C03650=1118.505,289.970,-75.818,-178.026,10.350,149.542
C03651=1118.509,289.721,-75.787,-178.029,10.347,149.543
C03652=1118.513,289.474,-75.756,-178.032,10.345,149.543
C03653=1118.517,289.225,-75.725,-178.035,10.342,149.543
C03654=1118.521,288.978,-75.694,-178.038,10.340,149.543
C03655=1118.526,288.730,-75.664,-178.041,10.338,149.543
C03656=1118.530,288.482,-75.632,-178.044,10.335,149.544
C03657=1118.534,288.234,-75.601,-178.047,10.333,149.544
C03658=1118.538,287.985,-75.570,-178.050,10.330,149.544
C03659=1118.542,287.738,-75.540,-178.053,10.327,149.544
C03660=1118.547,287.490,-75.509,-178.056,10.325,149.544
C03661=1118.551,287.241,-75.478,-178.060,10.322,149.544
C03662=1118.554,286.994,-75.447,-178.062,10.319,149.544
C03663=1118.558,286.745,-75.416,-178.065,10.318,149.545
C03664=1118.563,286.497,-75.385,-178.068,10.315,149.545
C03665=1118.568,286.249,-75.354,-178.071,10.313,149.545
C03666=1118.571,286.001,-75.324,-178.074,10.310,149.545
C03667=1118.576,285.753,-75.293,-178.077,10.307,149.545
C03668=1118.580,285.505,-75.262,-178.081,10.305,149.546
C03669=1118.583,285.257,-75.232,-178.084,10.302,149.546
C03670=1118.588,285.009,-75.201,-178.087,10.299,149.546
C03671=1118.593,284.761,-75.170,-178.090,10.297,149.546
C03672=1118.596,284.512,-75.140,-178.093,10.295,149.546
C03673=1118.601,284.264,-75.109,-178.096,10.292,149.546
C03674=1118.605,284.016,-75.078,-178.098,10.290,149.547
C03675=1118.608,283.768,-75.048,-178.102,10.287,149.547
C03676=1118.613,283.520,-75.017,-178.105,10.284,149.547
C03677=1118.617,283.273,-74.987,-178.108,10.282,149.547
C03678=1118.621,283.025,-74.956,-178.111,10.279,149.547
C03679=1118.626,282.776,-74.925,-178.114,10.277,149.548
C03680=1118.629,282.528,-74.895,-178.117,10.274,149.548
C03681=1118.634,282.280,-74.864,-178.120,10.272,149.548
C03682=1118.638,282.031,-74.834,-178.123,10.270,149.548
C03683=1118.642,281.783,-74.803,-178.126,10.267,149.548
C03684=1118.646,281.536,-74.773,-178.129,10.264,149.548
C03685=1118.650,281.323,-74.747,-178.132,10.262,149.549
C03686=1118.653,281.110,-74.721,-178.134,10.260,149.549
C03687=1118.657,280.897,-74.694,-178.138,10.257,149.549
C03688=1118.661,280.684,-74.668,-178.140,10.255,149.549
C03689=1118.664,280.471,-74.642,-178.143,10.252,149.549
C03690=1118.668,280.258,-74.616,-178.146,10.251,149.549
C03691=1118.671,280.045,-74.591,-178.149,10.248,149.550
C03692=1118.675,279.832,-74.564,-178.152,10.245,149.550
C03693=1118.679,279.584,-74.534,-178.155,10.243,149.550
C03694=1118.684,279.336,-74.503,-178.158,10.240,149.550
C03695=1118.687,279.087,-74.473,-178.161,10.237,149.550
C03696=1118.692,278.839,-74.443,-178.164,10.235,149.550
C03697=1118.696,278.591,-74.412,-178.167,10.232,149.551
C03698=1118.700,278.343,-74.383,-178.170,10.230,149.551
C03699=1118.705,278.095,-74.352,-178.173,10.227,149.551
C03700=1118.708,277.847,-74.322,-178.176,10.224,149.551
C03701=1118.713,277.598,-74.292,-178.180,10.222,149.551
C03702=1118.717,277.351,-74.262,-178.183,10.219,149.551
C03703=1118.721,277.102,-74.232,-178.186,10.216,149.551
C03704=1118.726,276.854,-74.201,-178.189,10.214,149.552
C03705=1118.730,276.606,-74.172,-178.192,10.211,149.552
C03706=1118.734,276.358,-74.142,-178.195,10.208,149.552
C03707=1118.738,276.109,-74.111,-178.198,10.205,149.552
C03708=1118.742,275.861,-74.081,-178.202,10.202,149.552
C03709=1118.746,275.613,-74.052,-178.205,10.200,149.552
C03710=1118.751,275.365,-74.021,-178.208,10.197,149.553
C03711=1118.755,275.117,-73.991,-178.210,10.195,149.553
C03712=1118.759,274.869,-73.961,-178.213,10.192,149.553
C03713=1118.763,274.621,-73.932,-178.216,10.190,149.553
C03714=1118.767,274.373,-73.901,-178.219,10.187,149.553
C03715=1118.771,274.124,-73.871,-178.222,10.184,149.553
C03716=1118.775,273.876,-73.842,-178.225,10.181,149.553
C03717=1118.779,273.628,-73.812,-178.228,10.179,149.553
C03718=1118.784,273.380,-73.782,-178.231,10.176,149.554
C03719=1118.788,273.132,-73.751,-178.234,10.173,149.554
C03720=1118.792,272.884,-73.722,-178.237,10.171,149.554
C03721=1118.796,272.635,-73.692,-178.240,10.168,149.554
C03722=1118.800,272.387,-73.663,-178.243,10.165,149.554
C03723=1118.805,272.139,-73.632,-178.245,10.163,149.554
C03724=1118.809,271.891,-73.603,-178.248,10.161,149.554
C03725=1118.813,271.643,-73.573,-178.251,10.158,149.554
C03726=1118.817,271.395,-73.543,-178.254,10.155,149.555
C03727=1118.822,271.147,-73.514,-178.257,10.152,149.555
C03728=1118.826,270.898,-73.484,-178.260,10.149,149.555
C03729=1118.831,270.650,-73.454,-178.262,10.148,149.555
C03730=1118.835,270.402,-73.425,-178.265,10.145,149.555
C03731=1118.839,270.154,-73.395,-178.268,10.142,149.555
C03732=1118.843,269.906,-73.365,-178.271,10.139,149.555
C03733=1118.847,269.657,-73.336,-178.274,10.136,149.555
C03734=1118.851,269.409,-73.306,-178.276,10.134,149.555
C03735=1118.855,269.161,-73.277,-178.279,10.132,149.555
C03736=1118.860,268.913,-73.247,-178.282,10.129,149.556
C03737=1118.864,268.664,-73.217,-178.285,10.126,149.556
C03738=1118.868,268.416,-73.187,-178.287,10.124,149.556
C03739=1118.873,268.168,-73.158,-178.290,10.121,149.556
C03740=1118.877,267.920,-73.128,-178.293,10.119,149.556
C03741=1118.880,267.707,-73.103,-178.296,10.117,149.556
C03742=1118.884,267.493,-73.078,-178.298,10.115,149.556
C03743=1118.888,267.281,-73.052,-178.300,10.113,149.556
C03744=1118.891,267.068,-73.027,-178.302,10.110,149.556
C03745=1118.895,266.854,-73.002,-178.304,10.108,149.556
C03746=1118.898,266.641,-72.977,-178.307,10.106,149.557
C03747=1118.903,266.428,-72.952,-178.310,10.104,149.557
C03748=1118.906,266.215,-72.926,-178.312,10.102,149.557
C03749=1118.910,265.967,-72.897,-178.314,10.100,149.557
C03750=1118.914,265.719,-72.867,-178.317,10.097,149.557
C03751=1118.918,265.470,-72.838,-178.320,10.095,149.557
C03752=1118.923,265.222,-72.809,-178.323,10.092,149.557
C03753=1118.927,264.973,-72.779,-178.325,10.090,149.557
C03754=1118.931,264.725,-72.750,-178.328,10.088,149.557
C03755=1118.935,264.477,-72.721,-178.331,10.085,149.558
C03756=1118.940,264.229,-72.692,-178.334,10.082,149.558
C03757=1118.944,263.981,-72.662,-178.337,10.080,149.558
C03758=1118.949,263.733,-72.633,-178.341,10.076,149.558
C03759=1118.952,263.485,-72.604,-178.344,10.074,149.558
C03760=1118.956,263.236,-72.575,-178.347,10.071,149.558
C03761=1118.961,262.988,-72.546,-178.350,10.067,149.559
C03762=1118.965,262.739,-72.516,-178.354,10.065,149.559
C03763=1118.970,262.492,-72.487,-178.357,10.062,149.559
C03764=1118.974,262.243,-72.458,-178.360,10.059,149.559
C03765=1118.978,261.995,-72.429,-178.364,10.056,149.559
C03766=1118.982,261.746,-72.399,-178.367,10.054,149.559
C03767=1118.986,261.498,-72.371,-178.370,10.050,149.560
C03768=1118.991,261.250,-72.342,-178.373,10.047,149.560
C03769=1118.995,261.002,-72.313,-178.376,10.044,149.560
C03770=1118.999,260.754,-72.283,-178.379,10.042,149.560
C03771=1119.004,260.505,-72.254,-178.382,10.039,149.560
C03772=1119.007,260.257,-72.226,-178.386,10.036,149.560
C03773=1119.012,260.009,-72.197,-178.389,10.033,149.560
C03774=1119.017,259.760,-72.168,-178.392,10.030,149.560
C03775=1119.021,259.512,-72.138,-178.395,10.027,149.561
C03776=1119.025,259.263,-72.110,-178.398,10.025,149.561
C03777=1119.029,259.015,-72.081,-178.401,10.022,149.561
C03778=1119.033,258.768,-72.052,-178.404,10.019,149.561
C03779=1119.038,258.519,-72.023,-178.407,10.016,149.561
C03780=1119.041,258.271,-71.994,-178.410,10.013,149.561
C03781=1119.046,258.022,-71.965,-178.413,10.010,149.561
C03782=1119.051,257.774,-71.936,-178.416,10.007,149.561
C03783=1119.054,257.526,-71.908,-178.418,10.004,149.561
C03784=1119.059,257.277,-71.879,-178.421,10.002,149.561
C03785=1119.064,257.029,-71.850,-178.424,9.999,149.561
C03786=1119.067,256.781,-71.822,-178.427,9.996,149.562
C03787=1119.072,256.532,-71.793,-178.430,9.993,149.561
C03788=1119.076,256.284,-71.764,-178.432,9.991,149.562
C03789=1119.080,256.036,-71.735,-178.435,9.988,149.562
C03790=1119.085,255.787,-71.707,-178.436,9.986,149.561
C03791=1119.088,255.539,-71.679,-178.437,9.985,149.561
C03792=1119.093,255.291,-71.649,-178.438,9.983,149.561
C03793=1119.098,255.042,-71.621,-178.439,9.981,149.561
C03794=1119.101,254.794,-71.592,-178.441,9.980,149.561
C03795=1119.106,254.546,-71.564,-178.442,9.977,149.561
C03796=1119.110,254.298,-71.535,-178.444,9.976,149.561
C03797=1119.114,254.084,-71.510,-178.445,9.974,149.561
C03798=1119.118,253.872,-71.485,-178.447,9.972,149.561
C03799=1119.121,253.658,-71.462,-178.449,9.971,149.561
C03800=1119.125,253.445,-71.437,-178.450,9.970,149.561
C03801=1119.129,253.231,-71.412,-178.452,9.967,149.561
C03802=1119.132,253.019,-71.388,-178.454,9.965,149.561
C03803=1119.136,252.805,-71.363,-178.457,9.963,149.561
C03804=1119.140,252.591,-71.338,-178.459,9.961,149.562
C03805=1119.144,252.344,-71.310,-178.461,9.959,149.562
C03806=1119.148,252.095,-71.281,-178.464,9.957,149.562
C03807=1119.153,251.847,-71.253,-178.468,9.954,149.562
C03808=1119.157,251.598,-71.225,-178.471,9.951,149.562
C03809=1119.161,251.350,-71.196,-178.474,9.949,149.563
C03810=1119.166,251.102,-71.167,-178.477,9.946,149.563
C03811=1119.169,250.854,-71.139,-178.481,9.943,149.563
C03812=1119.174,250.605,-71.110,-178.484,9.941,149.563
C03813=1119.178,250.357,-71.083,-178.488,9.937,149.564
C03814=1119.183,250.108,-71.054,-178.492,9.934,149.564
C03815=1119.187,249.860,-71.026,-178.496,9.931,149.564
C03816=1119.190,249.612,-70.997,-178.500,9.928,149.564
C03817=1119.196,249.364,-70.969,-178.504,9.924,149.564
C03818=1119.199,249.115,-70.941,-178.509,9.920,149.565
C03819=1119.204,248.866,-70.912,-178.513,9.917,149.565
C03820=1119.208,248.619,-70.884,-178.518,9.913,149.565
C03821=1119.212,248.370,-70.856,-178.523,9.909,149.566
C03822=1119.217,248.122,-70.828,-178.528,9.904,149.566
C03823=1119.221,247.873,-70.800,-178.533,9.900,149.566
C03824=1119.225,247.625,-70.772,-178.538,9.896,149.567
C03825=1119.230,247.376,-70.744,-178.542,9.892,149.567
C03826=1119.234,247.128,-70.716,-178.543,9.890,149.567
C03827=1119.238,246.879,-70.688,-178.545,9.887,149.567
C03828=1119.243,246.631,-70.660,-178.547,9.885,149.566
C03829=1119.247,246.383,-70.631,-178.549,9.883,149.566
C03830=1119.251,246.135,-70.604,-178.551,9.880,149.566
C03831=1119.255,245.886,-70.576,-178.553,9.878,149.566
C03832=1119.260,245.637,-70.548,-178.554,9.875,149.566
C03833=1119.264,245.389,-70.520,-178.557,9.872,149.566
C03834=1119.268,245.141,-70.492,-178.559,9.870,149.566
C03835=1119.273,244.893,-70.464,-178.561,9.868,149.566
C03836=1119.277,244.644,-70.435,-178.563,9.866,149.566
C03837=1119.282,244.396,-70.408,-178.565,9.863,149.566
C03838=1119.286,244.147,-70.380,-178.567,9.861,149.566
C03839=1119.290,243.899,-70.352,-178.569,9.858,149.566
C03840=1119.295,243.650,-70.324,-178.571,9.856,149.566
C03841=1119.299,243.402,-70.296,-178.573,9.853,149.566
C03842=1119.303,243.153,-70.268,-178.575,9.851,149.566
C03843=1119.307,242.905,-70.241,-178.578,9.848,149.566
C03844=1119.312,242.658,-70.213,-178.580,9.846,149.566
C03845=1119.316,242.408,-70.185,-178.582,9.844,149.566
C03846=1119.321,242.160,-70.157,-178.584,9.841,149.566
C03847=1119.325,241.912,-70.129,-178.587,9.839,149.566
C03848=1119.329,241.663,-70.102,-178.589,9.836,149.566
C03849=1119.334,241.415,-70.074,-178.591,9.834,149.566
C03850=1119.337,241.167,-70.046,-178.594,9.831,149.566
C03851=1119.342,240.918,-70.019,-178.596,9.829,149.566
C03852=1119.346,240.669,-69.990,-178.598,9.826,149.566
C03853=1119.350,240.456,-69.967,-178.601,9.824,149.566
C03854=1119.354,240.243,-69.943,-178.603,9.822,149.566
C03855=1119.357,240.029,-69.919,-178.605,9.820,149.566
C03856=1119.361,239.816,-69.895,-178.607,9.818,149.566
C03857=1119.365,239.603,-69.872,-178.609,9.816,149.566
C03858=1119.368,239.389,-69.848,-178.611,9.813,149.566
C03859=1119.372,239.176,-69.824,-178.613,9.811,149.566
C03860=1119.376,238.963,-69.801,-178.615,9.809,149.566
C03861=1119.381,238.714,-69.773,-178.618,9.807,149.566
C03862=1119.385,238.466,-69.745,-178.621,9.804,149.567
C03863=1119.390,238.217,-69.718,-178.624,9.802,149.567
C03864=1119.393,237.969,-69.690,-178.625,9.799,149.567
C03865=1119.398,237.720,-69.663,-178.628,9.796,149.567
C03866=1119.402,237.472,-69.635,-178.631,9.794,149.567
C03867=1119.406,237.223,-69.608,-178.634,9.792,149.567
C03868=1119.411,236.975,-69.581,-178.637,9.789,149.567
C03869=1119.415,236.727,-69.553,-178.639,9.786,149.567
C03870=1119.420,236.478,-69.526,-178.642,9.783,149.567
C03871=1119.424,236.230,-69.498,-178.644,9.781,149.567
C03872=1119.428,235.981,-69.470,-178.647,9.778,149.567
C03873=1119.433,235.733,-69.443,-178.650,9.776,149.568
C03874=1119.437,235.484,-69.415,-178.653,9.773,149.568
C03875=1119.442,235.236,-69.388,-178.656,9.770,149.568
C03876=1119.445,234.988,-69.362,-178.659,9.767,149.568
C03877=1119.450,234.740,-69.334,-178.662,9.764,149.568
C03878=1119.454,234.491,-69.307,-178.665,9.762,149.568
C03879=1119.459,234.242,-69.279,-178.667,9.759,149.568
C03880=1119.463,233.994,-69.252,-178.670,9.756,149.568
C03881=1119.468,233.746,-69.225,-178.673,9.753,149.568
C03882=1119.472,233.496,-69.197,-178.676,9.751,149.568
C03883=1119.476,233.248,-69.170,-178.679,9.748,149.569
C03884=1119.481,233.000,-69.142,-178.682,9.745,149.569
C03885=1119.485,232.752,-69.116,-178.685,9.742,149.569
C03886=1119.489,232.503,-69.088,-178.688,9.740,149.569
C03887=1119.493,232.254,-69.061,-178.691,9.736,149.569
C03888=1119.498,232.006,-69.034,-178.694,9.733,149.569
C03889=1119.503,231.757,-69.007,-178.697,9.730,149.569
C03890=1119.507,231.509,-68.980,-178.700,9.727,149.569
C03891=1119.510,231.260,-68.953,-178.704,9.724,149.569
C03892=1119.515,231.012,-68.926,-178.707,9.721,149.569
C03893=1119.520,230.763,-68.899,-178.710,9.718,149.570
C03894=1119.524,230.515,-68.872,-178.713,9.715,149.570
C03895=1119.528,230.267,-68.845,-178.716,9.712,149.570
C03896=1119.533,230.018,-68.818,-178.720,9.709,149.570
C03897=1119.537,229.770,-68.791,-178.723,9.706,149.570
C03898=1119.541,229.521,-68.763,-178.726,9.702,149.570
C03899=1119.545,229.272,-68.737,-178.729,9.699,149.570
C03900=1119.550,229.024,-68.710,-178.732,9.696,149.570
C03901=1119.555,228.775,-68.683,-178.735,9.693,149.570
C03902=1119.559,228.527,-68.656,-178.739,9.689,149.570
C03903=1119.563,228.279,-68.629,-178.741,9.686,149.570
C03904=1119.568,228.030,-68.602,-178.744,9.684,149.571
C03905=1119.573,227.782,-68.575,-178.748,9.680,149.571
C03906=1119.576,227.533,-68.548,-178.750,9.677,149.571
C03907=1119.581,227.284,-68.521,-178.754,9.673,149.571
C03908=1119.585,227.036,-68.496,-178.757,9.670,149.571
C03909=1119.589,226.823,-68.472,-178.759,9.668,149.571
C03910=1119.593,226.609,-68.449,-178.762,9.664,149.571
C03911=1119.597,226.395,-68.427,-178.764,9.662,149.571
C03912=1119.600,226.182,-68.403,-178.767,9.659,149.571
C03913=1119.604,225.969,-68.380,-178.769,9.656,149.571
C03914=1119.608,225.755,-68.358,-178.771,9.654,149.571
C03915=1119.612,225.542,-68.335,-178.774,9.651,149.571
C03916=1119.615,225.329,-68.312,-178.777,9.648,149.571
C03917=1119.620,225.079,-68.285,-178.779,9.645,149.571
C03918=1119.624,224.831,-68.259,-178.782,9.642,149.571
C03919=1119.628,224.582,-68.231,-178.785,9.639,149.571
C03920=1119.632,224.334,-68.205,-178.788,9.635,149.571
C03921=1119.637,224.085,-68.179,-178.790,9.632,149.571
C03922=1119.641,223.837,-68.152,-178.793,9.629,149.571
C03923=1119.646,223.588,-68.125,-178.796,9.626,149.571
C03924=1119.650,223.339,-68.099,-178.798,9.623,149.571
C03925=1119.655,223.091,-68.072,-178.802,9.619,149.571
C03926=1119.659,222.843,-68.046,-178.804,9.616,149.570
C03927=1119.664,222.594,-68.020,-178.807,9.613,149.570
C03928=1119.668,222.346,-67.993,-178.809,9.610,149.570
C03929=1119.673,222.097,-67.967,-178.812,9.607,149.570
C03930=1119.677,221.849,-67.941,-178.814,9.604,149.570
C03931=1119.682,221.600,-67.914,-178.817,9.601,149.570
C03932=1119.686,221.351,-67.888,-178.819,9.598,149.570
C03933=1119.690,221.103,-67.862,-178.822,9.594,149.570
C03934=1119.695,220.854,-67.835,-178.824,9.591,149.570
C03935=1119.699,220.606,-67.809,-178.827,9.588,149.570
C03936=1119.704,220.357,-67.782,-178.829,9.585,149.570
C03937=1119.708,220.108,-67.756,-178.832,9.582,149.570
C03938=1119.712,219.860,-67.730,-178.834,9.578,149.569
C03939=1119.717,219.611,-67.704,-178.837,9.575,149.569
C03940=1119.721,219.363,-67.677,-178.839,9.572,149.569
C03941=1119.725,219.114,-67.651,-178.842,9.569,149.569
C03942=1119.730,218.866,-67.625,-178.844,9.567,149.569
C03943=1119.734,218.617,-67.599,-178.846,9.564,149.569
C03944=1119.739,218.368,-67.573,-178.848,9.560,149.569
C03945=1119.743,218.120,-67.546,-178.851,9.557,149.569
C03946=1119.748,217.871,-67.520,-178.853,9.554,149.569
C03947=1119.751,217.623,-67.494,-178.855,9.552,149.569
C03948=1119.756,217.374,-67.468,-178.857,9.548,149.568
C03949=1119.761,217.125,-67.442,-178.860,9.545,149.568
C03950=1119.765,216.877,-67.415,-178.862,9.543,149.568
C03951=1119.769,216.629,-67.390,-178.864,9.539,149.568
C03952=1119.774,216.379,-67.364,-178.866,9.536,149.568
C03953=1119.779,216.131,-67.338,-178.868,9.534,149.568
C03954=1119.782,215.883,-67.311,-178.871,9.531,149.568
C03955=1119.787,215.634,-67.286,-178.873,9.527,149.568
C03956=1119.792,215.385,-67.259,-178.875,9.525,149.568
C03957=1119.796,215.136,-67.234,-178.877,9.522,149.568
C03958=1119.800,214.888,-67.207,-178.879,9.519,149.567
C03959=1119.805,214.639,-67.182,-178.881,9.516,149.567
C03960=1119.809,214.391,-67.156,-178.883,9.513,149.567
C03961=1119.814,214.142,-67.130,-178.885,9.510,149.567
C03962=1119.819,213.893,-67.104,-178.887,9.508,149.567
C03963=1119.823,213.645,-67.078,-178.889,9.505,149.567
C03964=1119.827,213.396,-67.052,-178.891,9.502,149.567
C03965=1119.831,213.114,-67.023,-178.894,9.499,149.567
C03966=1119.838,212.832,-66.994,-178.896,9.496,149.566
C03967=1119.842,212.550,-66.964,-178.899,9.493,149.566
C03968=1119.847,212.267,-66.935,-178.902,9.489,149.566
C03969=1119.851,212.019,-66.909,-178.904,9.487,149.566
C03970=1119.856,211.770,-66.883,-178.906,9.483,149.566
C03971=1119.861,211.521,-66.857,-178.909,9.480,149.566
C03972=1119.865,211.272,-66.832,-178.911,9.478,149.566
C03973=1119.870,211.024,-66.806,-178.913,9.475,149.566
C03974=1119.874,210.775,-66.780,-178.916,9.472,149.566
C03975=1119.878,210.526,-66.755,-178.919,9.469,149.566
C03976=1119.882,210.278,-66.729,-178.921,9.467,149.566
C03977=1119.887,210.030,-66.704,-178.923,9.464,149.566
C03978=1119.891,209.781,-66.678,-178.926,9.461,149.566
C03979=1119.896,209.532,-66.652,-178.929,9.458,149.566
C03980=1119.900,209.284,-66.627,-178.931,9.455,149.566
C03981=1119.905,209.035,-66.601,-178.933,9.453,149.566
C03982=1119.909,208.786,-66.575,-178.936,9.450,149.566
C03983=1119.914,208.538,-66.550,-178.939,9.447,149.566
C03984=1119.918,208.289,-66.524,-178.941,9.444,149.566
C03985=1119.925,207.896,-66.483,-178.946,9.439,149.566
C03986=1119.932,207.502,-66.442,-178.950,9.435,149.566
C03987=1119.940,207.108,-66.403,-178.955,9.430,149.567
C03988=1119.947,206.715,-66.362,-178.959,9.426,149.567
C03989=1119.951,206.466,-66.336,-178.962,9.423,149.567
C03990=1119.956,206.218,-66.311,-178.964,9.420,149.567
C03991=1119.960,205.969,-66.286,-178.967,9.417,149.567
C03992=1119.964,205.720,-66.261,-178.970,9.414,149.567
C03993=1119.969,205.472,-66.235,-178.973,9.412,149.567
C03994=1119.973,205.223,-66.209,-178.976,9.409,149.567
C03995=1119.977,204.973,-66.184,-178.979,9.406,149.567
C03996=1119.982,204.725,-66.159,-178.982,9.403,149.567
C03997=1119.987,204.477,-66.133,-178.985,9.400,149.568
C03998=1119.992,204.228,-66.109,-178.987,9.397,149.568
C03999=1119.996,203.979,-66.083,-178.990,9.394,149.568
C04000=1120.000,203.731,-66.058,-178.993,9.392,149.568
C04001=1120.004,203.482,-66.033,-178.997,9.388,149.568
C04002=1120.009,203.233,-66.007,-178.999,9.385,149.568
C04003=1120.014,202.985,-65.982,-179.002,9.382,149.568
C04004=1120.018,202.735,-65.957,-179.005,9.380,149.568
C04005=1120.023,202.487,-65.931,-179.008,9.377,149.568
C04006=1120.027,202.238,-65.907,-179.012,9.373,149.568
C04007=1120.032,201.990,-65.882,-179.014,9.370,149.568
C04008=1120.036,201.741,-65.857,-179.017,9.368,149.569
C04009=1120.041,201.493,-65.831,-179.021,9.364,149.569
C04010=1120.045,201.243,-65.807,-179.024,9.361,149.569
C04011=1120.049,200.995,-65.781,-179.026,9.359,149.569
C04012=1120.054,200.746,-65.756,-179.030,9.355,149.569
C04013=1120.058,200.497,-65.731,-179.033,9.352,149.569
C04014=1120.063,200.249,-65.707,-179.036,9.349,149.569
C04015=1120.067,200.000,-65.681,-179.039,9.346,149.569
C04016=1120.072,199.751,-65.656,-179.042,9.343,149.569
C04017=1120.076,199.537,-65.635,-179.045,9.340,149.569
C04018=1120.080,199.324,-65.614,-179.048,9.337,149.570
C04019=1120.083,199.110,-65.592,-179.050,9.334,149.570
C04020=1120.087,198.896,-65.571,-179.053,9.331,149.570
C04021=1120.091,198.683,-65.549,-179.056,9.328,149.570
C04022=1120.095,198.469,-65.528,-179.059,9.325,149.570
C04023=1120.098,198.255,-65.506,-179.061,9.323,149.570
C04024=1120.103,198.042,-65.485,-179.064,9.319,149.570
C04025=1120.107,197.793,-65.460,-179.067,9.317,149.570
C04026=1120.111,197.544,-65.436,-179.071,9.313,149.570
C04027=1120.116,197.295,-65.411,-179.074,9.309,149.570
C04028=1120.120,197.047,-65.386,-179.077,9.306,149.570
C04029=1120.125,196.798,-65.361,-179.080,9.303,149.570
C04030=1120.130,196.549,-65.336,-179.083,9.299,149.570
C04031=1120.134,196.301,-65.312,-179.087,9.295,149.570
C04032=1120.138,196.051,-65.287,-179.088,9.293,149.570
C04033=1120.143,195.803,-65.263,-179.090,9.290,149.570
C04034=1120.148,195.555,-65.237,-179.092,9.288,149.570
C04035=1120.151,195.306,-65.213,-179.093,9.285,149.570
C04036=1120.157,195.057,-65.188,-179.096,9.282,149.570
C04037=1120.160,194.808,-65.164,-179.097,9.279,149.569
C04038=1120.166,194.559,-65.139,-179.099,9.277,149.569
C04039=1120.170,194.311,-65.115,-179.101,9.275,149.569
C04040=1120.174,194.061,-65.090,-179.103,9.271,149.569
C04041=1120.179,193.813,-65.066,-179.105,9.269,149.569
C04042=1120.184,193.565,-65.041,-179.107,9.266,149.569
C04043=1120.187,193.316,-65.016,-179.109,9.263,149.569
C04044=1120.193,193.067,-64.992,-179.111,9.261,149.569
C04045=1120.197,192.818,-64.967,-179.113,9.259,149.569
C04046=1120.202,192.569,-64.942,-179.115,9.255,149.568
C04047=1120.206,192.321,-64.918,-179.117,9.253,149.568
C04048=1120.210,192.072,-64.894,-179.119,9.250,149.568
C04049=1120.215,191.823,-64.869,-179.121,9.247,149.568
C04050=1120.219,191.574,-64.845,-179.123,9.245,149.568
C04051=1120.224,191.326,-64.821,-179.125,9.242,149.568
C04052=1120.228,191.077,-64.796,-179.127,9.239,149.568
C04053=1120.233,190.828,-64.772,-179.129,9.237,149.568
C04054=1120.238,190.579,-64.747,-179.132,9.234,149.568
C04055=1120.242,190.331,-64.723,-179.133,9.231,149.568
C04056=1120.247,190.082,-64.698,-179.136,9.228,149.568
C04057=1120.251,189.833,-64.674,-179.138,9.226,149.568
C04058=1120.256,189.584,-64.651,-179.140,9.223,149.568
C04059=1120.261,189.335,-64.626,-179.142,9.220,149.568
C04060=1120.265,189.086,-64.602,-179.145,9.217,149.568
C04061=1120.269,188.838,-64.578,-179.147,9.214,149.568
C04062=1120.274,188.589,-64.553,-179.149,9.212,149.568
C04063=1120.278,188.340,-64.528,-179.152,9.209,149.568
C04064=1120.282,188.092,-64.504,-179.154,9.206,149.568
C04065=1120.288,187.842,-64.480,-179.156,9.203,149.567
C04066=1120.292,187.594,-64.456,-179.159,9.200,149.567
C04067=1120.297,187.345,-64.432,-179.161,9.198,149.567
C04068=1120.301,187.096,-64.407,-179.163,9.195,149.567
C04069=1120.306,186.848,-64.383,-179.166,9.192,149.567
C04070=1120.310,186.599,-64.360,-179.167,9.189,149.567
C04071=1120.315,186.350,-64.336,-179.170,9.186,149.567
C04072=1120.319,186.101,-64.311,-179.173,9.183,149.567
C04073=1120.323,185.887,-64.291,-179.174,9.181,149.567
C04074=1120.327,185.674,-64.270,-179.176,9.179,149.567
C04075=1120.331,185.459,-64.249,-179.179,9.175,149.567
C04076=1120.335,185.246,-64.228,-179.181,9.173,149.567
C04077=1120.338,185.032,-64.208,-179.183,9.171,149.567
C04078=1120.343,184.818,-64.187,-179.186,9.168,149.567
C04079=1120.347,184.604,-64.166,-179.187,9.166,149.567
C04080=1120.350,184.390,-64.146,-179.189,9.163,149.567
C04081=1120.355,184.142,-64.122,-179.192,9.160,149.567
C04082=1120.360,183.893,-64.097,-179.194,9.157,149.567
C04083=1120.364,183.644,-64.074,-179.197,9.154,149.567
C04084=1120.368,183.395,-64.050,-179.200,9.151,149.567
C04085=1120.373,183.146,-64.026,-179.202,9.148,149.567
C04086=1120.377,182.898,-64.002,-179.205,9.145,149.567
C04087=1120.382,182.649,-63.978,-179.207,9.142,149.567
C04088=1120.387,182.400,-63.955,-179.210,9.139,149.567
C04089=1120.392,182.152,-63.930,-179.213,9.136,149.567
C04090=1120.396,181.902,-63.907,-179.215,9.133,149.567
C04091=1120.400,181.653,-63.882,-179.218,9.130,149.567
C04092=1120.405,181.404,-63.859,-179.221,9.126,149.567
C04093=1120.409,181.156,-63.835,-179.224,9.123,149.567
C04094=1120.414,180.907,-63.811,-179.226,9.120,149.567
C04095=1120.418,180.658,-63.787,-179.229,9.117,149.567
C04096=1120.423,180.409,-63.764,-179.231,9.114,149.567
C04097=1120.427,180.161,-63.740,-179.234,9.110,149.567
C04098=1120.432,179.912,-63.717,-179.237,9.107,149.567
C04099=1120.437,179.663,-63.693,-179.240,9.104,149.567
C04100=1120.441,179.415,-63.669,-179.242,9.101,149.567
C04101=1120.446,179.166,-63.646,-179.245,9.098,149.567
C04102=1120.451,178.916,-63.622,-179.247,9.094,149.567
C04103=1120.454,178.667,-63.598,-179.250,9.091,149.566
C04104=1120.459,178.418,-63.575,-179.251,9.089,149.566
C04105=1120.464,178.170,-63.551,-179.254,9.085,149.566
C04106=1120.468,177.921,-63.527,-179.255,9.083,149.566
C04107=1120.473,177.672,-63.504,-179.258,9.080,149.566
C04108=1120.478,177.423,-63.480,-179.260,9.076,149.566
C04109=1120.482,177.174,-63.456,-179.262,9.074,149.566
C04110=1120.487,176.925,-63.433,-179.264,9.071,149.566
C04111=1120.491,176.676,-63.410,-179.267,9.067,149.566
C04112=1120.496,176.428,-63.386,-179.268,9.065,149.566
C04113=1120.501,176.179,-63.362,-179.271,9.062,149.566
C04114=1120.504,175.930,-63.339,-179.273,9.058,149.565
C04115=1120.509,175.681,-63.316,-179.275,9.056,149.565
C04116=1120.514,175.432,-63.293,-179.277,9.053,149.565
C04117=1120.518,175.184,-63.269,-179.280,9.050,149.565
C04118=1120.523,174.935,-63.245,-179.281,9.047,149.565
C04119=1120.528,174.686,-63.222,-179.284,9.044,149.565
C04120=1120.532,174.437,-63.199,-179.286,9.041,149.565
C04121=1120.537,174.188,-63.175,-179.288,9.038,149.565
C04122=1120.542,173.940,-63.153,-179.290,9.035,149.565
C04123=1120.546,173.691,-63.129,-179.293,9.032,149.565
C04124=1120.551,173.442,-63.105,-179.294,9.029,149.564
C04125=1120.555,173.193,-63.082,-179.297,9.026,149.564
C04126=1120.560,172.944,-63.059,-179.300,9.023,149.564
C04127=1120.565,172.695,-63.035,-179.302,9.020,149.564
C04128=1120.569,172.446,-63.013,-179.304,9.017,149.564
C04129=1120.573,172.232,-62.992,-179.305,9.015,149.564
C04130=1120.576,172.018,-62.972,-179.308,9.012,149.564
C04131=1120.581,171.804,-62.953,-179.309,9.009,149.564
C04132=1120.585,171.590,-62.933,-179.311,9.007,149.564
C04133=1120.589,171.377,-62.913,-179.313,9.005,149.564
C04134=1120.593,171.163,-62.893,-179.316,9.001,149.564
C04135=1120.597,170.948,-62.872,-179.317,8.999,149.563
C04136=1120.601,170.734,-62.853,-179.319,8.996,149.563
C04137=1120.605,170.485,-62.830,-179.322,8.993,149.563
C04138=1120.609,170.236,-62.807,-179.324,8.990,149.563
C04139=1120.615,169.988,-62.784,-179.326,8.987,149.563
C04140=1120.619,169.739,-62.761,-179.328,8.984,149.563
C04141=1120.624,169.490,-62.737,-179.331,8.981,149.563
C04142=1120.628,169.241,-62.714,-179.333,8.978,149.563
C04143=1120.633,168.992,-62.691,-179.335,8.975,149.563
C04144=1120.637,168.743,-62.668,-179.337,8.972,149.563
C04145=1120.641,168.495,-62.645,-179.339,8.969,149.562
C04146=1120.647,168.246,-62.622,-179.342,8.966,149.562
C04147=1120.652,167.997,-62.599,-179.344,8.963,149.562
C04148=1120.656,167.748,-62.577,-179.346,8.960,149.562
C04149=1120.660,167.499,-62.553,-179.348,8.957,149.562
C04150=1120.665,167.250,-62.530,-179.351,8.954,149.562
C04151=1120.670,167.002,-62.507,-179.353,8.951,149.562
C04152=1120.675,166.752,-62.485,-179.355,8.947,149.562
C04153=1120.679,166.503,-62.462,-179.358,8.944,149.562
C04154=1120.683,166.254,-62.439,-179.360,8.942,149.562
C04155=1120.688,166.005,-62.415,-179.362,8.938,149.561
C04156=1120.693,165.757,-62.394,-179.364,8.935,149.561
C04157=1120.697,165.508,-62.370,-179.367,8.932,149.561
C04158=1120.701,165.259,-62.348,-179.369,8.928,149.561
C04159=1120.706,165.010,-62.324,-179.372,8.925,149.561
C04160=1120.711,164.761,-62.303,-179.374,8.922,149.561
C04161=1120.716,164.512,-62.279,-179.376,8.919,149.561
C04162=1120.720,164.263,-62.256,-179.379,8.916,149.561
C04163=1120.725,164.014,-62.234,-179.381,8.913,149.561
C04164=1120.730,163.766,-62.211,-179.383,8.910,149.560
C04165=1120.734,163.517,-62.188,-179.385,8.907,149.560
C04166=1120.739,163.267,-62.165,-179.388,8.904,149.560
C04167=1120.743,163.018,-62.143,-179.390,8.900,149.560
C04168=1120.748,162.770,-62.121,-179.392,8.897,149.560
C04169=1120.752,162.521,-62.098,-179.395,8.894,149.560
C04170=1120.757,162.271,-62.075,-179.397,8.890,149.560
C04171=1120.761,162.022,-62.052,-179.399,8.887,149.560
C04172=1120.766,161.774,-62.030,-179.401,8.884,149.560
C04173=1120.771,161.525,-62.007,-179.404,8.881,149.560
C04174=1120.775,161.276,-61.984,-179.407,8.878,149.560
C04175=1120.781,161.027,-61.962,-179.409,8.874,149.559
C04176=1120.785,160.778,-61.939,-179.411,8.871,149.559
C04177=1120.789,160.529,-61.917,-179.413,8.868,149.559
C04178=1120.794,160.281,-61.894,-179.416,8.864,149.559
C04179=1120.798,160.031,-61.872,-179.418,8.861,149.559
C04180=1120.803,159.782,-61.850,-179.420,8.858,149.559
C04181=1120.808,159.534,-61.827,-179.423,8.855,149.559
C04182=1120.812,159.284,-61.805,-179.425,8.851,149.558
C04183=1120.817,159.035,-61.782,-179.427,8.848,149.558
C04184=1120.822,158.787,-61.760,-179.430,8.845,149.558
C04185=1120.826,158.572,-61.741,-179.431,8.842,149.558
C04186=1120.830,158.358,-61.722,-179.434,8.839,149.558
C04187=1120.834,158.145,-61.702,-179.435,8.837,149.558
C04188=1120.838,157.930,-61.683,-179.438,8.833,149.558
C04189=1120.842,157.716,-61.664,-179.439,8.831,149.558
C04190=1120.846,157.502,-61.645,-179.442,8.828,149.558
C04191=1120.850,157.288,-61.626,-179.444,8.824,149.558
C04192=1120.853,157.075,-61.607,-179.446,8.822,149.557
C04193=1120.858,156.825,-61.584,-179.448,8.819,149.557
C04194=1120.863,156.576,-61.562,-179.451,8.815,149.557
C04195=1120.867,156.327,-61.540,-179.453,8.812,149.557
C04196=1120.872,156.078,-61.517,-179.456,8.808,149.557
C04197=1120.877,155.829,-61.495,-179.458,8.805,149.557
C04198=1120.881,155.580,-61.473,-179.460,8.801,149.557
C04199=1120.886,155.331,-61.451,-179.462,8.798,149.556
C04200=1120.890,155.082,-61.429,-179.465,8.795,149.556
C04201=1120.896,154.834,-61.406,-179.467,8.791,149.556
C04202=1120.900,154.584,-61.384,-179.470,8.788,149.556
C04203=1120.905,154.336,-61.363,-179.472,8.784,149.556
C04204=1120.909,154.086,-61.341,-179.475,8.781,149.556
C04205=1120.914,153.838,-61.319,-179.477,8.777,149.556
C04206=1120.919,153.588,-61.296,-179.479,8.774,149.555
C04207=1120.924,153.339,-61.275,-179.481,8.771,149.555
C04208=1120.928,153.091,-61.252,-179.484,8.766,149.555
C04209=1120.932,152.842,-61.230,-179.487,8.763,149.555
C04210=1120.937,152.593,-61.208,-179.489,8.760,149.555
C04211=1120.942,152.344,-61.186,-179.491,8.756,149.555
C04212=1120.946,152.095,-61.164,-179.494,8.752,149.554
C04213=1120.952,151.846,-61.142,-179.496,8.749,149.554
C04214=1120.956,151.596,-61.120,-179.498,8.745,149.554
C04215=1120.961,151.348,-61.098,-179.501,8.742,149.554
C04216=1120.965,151.099,-61.076,-179.503,8.738,149.554
C04217=1120.970,150.850,-61.055,-179.505,8.734,149.554
C04218=1120.974,150.601,-61.033,-179.508,8.731,149.553
C04219=1120.979,150.352,-61.011,-179.511,8.727,149.553
C04220=1120.983,150.103,-60.989,-179.513,8.724,149.553
C04221=1120.988,149.853,-60.968,-179.515,8.720,149.553
C04222=1120.993,149.605,-60.946,-179.518,8.716,149.553
C04223=1120.998,149.355,-60.924,-179.520,8.713,149.553
C04224=1121.002,149.107,-60.902,-179.522,8.709,149.552
C04225=1121.007,148.857,-60.880,-179.525,8.705,149.552
C04226=1121.012,148.609,-60.859,-179.527,8.702,149.552
C04227=1121.016,148.360,-60.837,-179.529,8.698,149.552
C04228=1121.021,148.110,-60.816,-179.532,8.694,149.552
C04229=1121.026,147.861,-60.794,-179.534,8.691,149.551
C04230=1121.030,147.612,-60.772,-179.537,8.686,149.551
C04231=1121.035,147.363,-60.750,-179.539,8.683,149.551
C04232=1121.040,147.115,-60.729,-179.542,8.679,149.551
C04233=1121.044,146.865,-60.707,-179.544,8.675,149.550
C04234=1121.049,146.616,-60.686,-179.546,8.672,149.550
C04235=1121.054,146.368,-60.664,-179.549,8.667,149.550
C04236=1121.058,146.118,-60.642,-179.551,8.664,149.550
C04237=1121.063,145.869,-60.621,-179.553,8.660,149.549
C04238=1121.068,145.621,-60.600,-179.556,8.657,149.549
C04239=1121.072,145.371,-60.578,-179.559,8.652,149.549
C04240=1121.077,145.122,-60.557,-179.561,8.649,149.549
C04241=1121.081,144.908,-60.538,-179.562,8.646,149.548
C04242=1121.085,144.694,-60.520,-179.563,8.643,149.548
C04243=1121.090,144.480,-60.501,-179.564,8.640,149.548
C04244=1121.093,144.265,-60.483,-179.566,8.637,149.548
C04245=1121.097,144.051,-60.464,-179.568,8.634,149.547
C04246=1121.101,143.837,-60.446,-179.569,8.631,149.547
C04247=1121.106,143.623,-60.428,-179.570,8.628,149.547
C04248=1121.109,143.409,-60.409,-179.572,8.625,149.546
C04249=1121.114,143.160,-60.388,-179.573,8.622,149.546
C04250=1121.118,142.911,-60.366,-179.575,8.619,149.546
C04251=1121.124,142.661,-60.345,-179.576,8.615,149.545
C04252=1121.128,142.413,-60.324,-179.577,8.612,149.545
C04253=1121.133,142.164,-60.303,-179.579,8.609,149.545
C04254=1121.137,141.915,-60.281,-179.581,8.605,149.544
C04255=1121.142,141.665,-60.260,-179.583,8.602,149.544
C04256=1121.147,141.417,-60.239,-179.584,8.598,149.544
C04257=1121.151,141.167,-60.218,-179.586,8.595,149.543
C04258=1121.156,140.918,-60.196,-179.587,8.592,149.543
C04259=1121.161,140.669,-60.175,-179.589,8.588,149.543
C04260=1121.166,140.420,-60.154,-179.590,8.585,149.542
C04261=1121.170,140.172,-60.133,-179.592,8.582,149.542
C04262=1121.175,139.922,-60.111,-179.593,8.578,149.542
C04263=1121.180,139.673,-60.090,-179.595,8.575,149.541
C04264=1121.184,139.424,-60.070,-179.597,8.572,149.541
C04265=1121.189,139.175,-60.048,-179.598,8.569,149.541
C04266=1121.194,138.925,-60.027,-179.600,8.565,149.541
C04267=1121.198,138.677,-60.006,-179.601,8.562,149.540
C04268=1121.203,138.428,-59.985,-179.603,8.559,149.540
C04269=1121.208,138.179,-59.964,-179.605,8.555,149.539
C04270=1121.212,137.930,-59.943,-179.606,8.552,149.539
C04271=1121.217,137.680,-59.921,-179.608,8.548,149.539
C04272=1121.222,137.431,-59.900,-179.609,8.545,149.539
C04273=1121.226,137.183,-59.879,-179.611,8.542,149.538
C04274=1121.231,136.933,-59.858,-179.612,8.539,149.538
C04275=1121.236,136.684,-59.838,-179.614,8.535,149.538
C04276=1121.241,136.436,-59.816,-179.617,8.532,149.537
C04277=1121.245,136.186,-59.795,-179.618,8.529,149.537
C04278=1121.250,135.937,-59.775,-179.620,8.525,149.537
C04279=1121.255,135.688,-59.754,-179.621,8.522,149.536
C04280=1121.259,135.439,-59.732,-179.623,8.519,149.536
C04281=1121.264,135.190,-59.712,-179.625,8.515,149.536
C04282=1121.269,134.941,-59.691,-179.626,8.512,149.535
C04283=1121.274,134.692,-59.670,-179.628,8.509,149.535
C04284=1121.279,134.443,-59.648,-179.629,8.506,149.535
C04285=1121.283,134.194,-59.628,-179.631,8.502,149.535
C04286=1121.288,133.944,-59.607,-179.633,8.499,149.534
C04287=1121.292,133.695,-59.586,-179.634,8.496,149.534
C04288=1121.297,133.446,-59.565,-179.636,8.492,149.534
C04289=1121.302,133.197,-59.545,-179.638,8.488,149.533
C04290=1121.307,132.948,-59.523,-179.640,8.486,149.533
C04291=1121.311,132.700,-59.503,-179.641,8.482,149.533
C04292=1121.316,132.450,-59.482,-179.643,8.479,149.533
C04293=1121.321,132.201,-59.462,-179.645,8.476,149.532
C04294=1121.326,131.952,-59.441,-179.646,8.472,149.532
C04295=1121.330,131.703,-59.420,-179.648,8.469,149.532
C04296=1121.335,131.453,-59.399,-179.650,8.466,149.531
C04297=1121.339,131.239,-59.382,-179.651,8.463,149.531
C04298=1121.343,131.025,-59.364,-179.653,8.460,149.531
C04299=1121.348,130.811,-59.346,-179.654,8.457,149.531
C04300=1121.351,130.596,-59.328,-179.655,8.454,149.530
C04301=1121.356,130.382,-59.311,-179.657,8.451,149.530
C04302=1121.359,130.168,-59.293,-179.659,8.448,149.530
C04303=1121.363,129.953,-59.275,-179.660,8.445,149.530
C04304=1121.368,129.739,-59.257,-179.662,8.443,149.529
C04305=1121.372,129.490,-59.237,-179.664,8.439,149.529
C04306=1121.378,129.241,-59.216,-179.665,8.436,149.529
C04307=1121.382,128.992,-59.195,-179.667,8.433,149.529
C04308=1121.386,128.743,-59.175,-179.669,8.429,149.528
C04309=1121.392,128.494,-59.154,-179.670,8.426,149.528
C04310=1121.396,128.245,-59.134,-179.672,8.423,149.528
C04311=1121.400,127.996,-59.113,-179.673,8.420,149.527
C04312=1121.406,127.747,-59.092,-179.675,8.416,149.527
C04313=1121.410,127.498,-59.072,-179.678,8.413,149.527
C04314=1121.415,127.249,-59.051,-179.679,8.409,149.527
C04315=1121.420,127.000,-59.031,-179.681,8.406,149.526
C04316=1121.424,126.750,-59.011,-179.683,8.403,149.526
C04317=1121.429,126.501,-58.991,-179.685,8.399,149.526
C04318=1121.434,126.252,-58.970,-179.686,8.396,149.525
C04319=1121.438,126.003,-58.949,-179.688,8.393,149.525
C04320=1121.443,125.754,-58.929,-179.690,8.389,149.525
C04321=1121.448,125.505,-58.908,-179.691,8.386,149.525
C04322=1121.453,125.255,-58.888,-179.693,8.383,149.524
C04323=1121.457,125.006,-58.868,-179.695,8.379,149.524
C04324=1121.462,124.757,-58.847,-179.696,8.376,149.524
C04325=1121.467,124.508,-58.827,-179.698,8.373,149.524
C04326=1121.472,124.258,-58.807,-179.701,8.369,149.523
C04327=1121.476,124.010,-58.787,-179.702,8.366,149.523
C04328=1121.481,123.761,-58.766,-179.704,8.363,149.523
C04329=1121.486,123.512,-58.746,-179.706,8.359,149.523
C04330=1121.491,123.262,-58.726,-179.708,8.356,149.522
C04331=1121.495,123.013,-58.706,-179.709,8.353,149.522
C04332=1121.500,122.765,-58.685,-179.711,8.349,149.522
C04333=1121.505,122.515,-58.665,-179.713,8.346,149.521
C04334=1121.510,122.266,-58.645,-179.715,8.342,149.521
C04335=1121.514,122.017,-58.624,-179.716,8.339,149.521
C04336=1121.519,121.767,-58.604,-179.718,8.336,149.521
C04337=1121.523,121.518,-58.584,-179.720,8.332,149.520
C04338=1121.528,121.270,-58.564,-179.722,8.329,149.520
C04339=1121.533,121.020,-58.544,-179.724,8.326,149.520
C04340=1121.538,120.771,-58.523,-179.725,8.322,149.519
C04341=1121.543,120.522,-58.504,-179.727,8.319,149.519
C04342=1121.548,120.273,-58.483,-179.729,8.315,149.519
C04343=1121.552,120.024,-58.463,-179.731,8.312,149.519
C04344=1121.557,119.774,-58.443,-179.733,8.309,149.519
C04345=1121.562,119.526,-58.423,-179.734,8.305,149.518
C04346=1121.567,119.276,-58.404,-179.737,8.301,149.518
C04347=1121.571,119.027,-58.383,-179.738,8.299,149.518
C04348=1121.576,118.778,-58.364,-179.740,8.295,149.517
C04349=1121.581,118.529,-58.343,-179.742,8.292,149.517
C04350=1121.586,118.279,-58.323,-179.744,8.288,149.517
C04351=1121.591,118.031,-58.303,-179.745,8.285,149.517
C04352=1121.595,117.781,-58.283,-179.747,8.282,149.516
C04353=1121.599,117.567,-58.266,-179.749,8.278,149.516
C04354=1121.604,117.352,-58.249,-179.751,8.275,149.516
C04355=1121.607,117.139,-58.232,-179.752,8.273,149.516
C04356=1121.611,116.924,-58.215,-179.754,8.270,149.515
C04357=1121.615,116.710,-58.198,-179.756,8.266,149.515
C04358=1121.619,116.495,-58.181,-179.757,8.264,149.515
C04359=1121.624,116.281,-58.163,-179.758,8.261,149.515
C04360=1121.628,116.067,-58.147,-179.760,8.257,149.514
C04361=1121.633,115.817,-58.127,-179.762,8.254,149.514
C04362=1121.637,115.568,-58.106,-179.764,8.251,149.514
C04363=1121.642,115.318,-58.087,-179.766,8.247,149.514
C04364=1121.647,115.070,-58.068,-179.767,8.244,149.513
C04365=1121.652,114.821,-58.047,-179.769,8.240,149.513
C04366=1121.657,114.571,-58.028,-179.771,8.237,149.513
C04367=1121.662,114.322,-58.008,-179.773,8.234,149.513
C04368=1121.666,114.073,-57.988,-179.774,8.230,149.512
C04369=1121.671,113.824,-57.968,-179.777,8.226,149.512
C04370=1121.676,113.574,-57.949,-179.779,8.223,149.512
C04371=1121.680,113.326,-57.930,-179.781,8.219,149.511
C04372=1121.685,113.077,-57.909,-179.782,8.216,149.511
C04373=1121.690,112.827,-57.890,-179.784,8.212,149.511
C04374=1121.695,112.578,-57.871,-179.786,8.209,149.511
C04375=1121.700,112.329,-57.851,-179.788,8.206,149.510
C04376=1121.704,112.080,-57.831,-179.789,8.202,149.510
C04377=1121.709,111.831,-57.811,-179.792,8.198,149.510
C04378=1121.714,111.581,-57.792,-179.794,8.195,149.509
C04379=1121.719,111.332,-57.772,-179.796,8.191,149.509
C04380=1121.724,111.083,-57.753,-179.797,8.188,149.509
C04381=1121.728,110.834,-57.734,-179.799,8.184,149.509
C04382=1121.733,110.585,-57.713,-179.801,8.181,149.508
C04383=1121.738,110.336,-57.694,-179.804,8.176,149.508
C04384=1121.743,110.086,-57.674,-179.806,8.173,149.508
C04385=1121.748,109.837,-57.655,-179.809,8.169,149.508
C04386=1121.752,109.588,-57.636,-179.811,8.165,149.507
C04387=1121.757,109.338,-57.616,-179.813,8.162,149.507
C04388=1121.762,109.089,-57.597,-179.816,8.157,149.507
C04389=1121.767,108.840,-57.577,-179.818,8.154,149.507
C04390=1121.771,108.591,-57.558,-179.820,8.149,149.507
C04391=1121.776,108.342,-57.539,-179.822,8.146,149.506
C04392=1121.781,108.092,-57.519,-179.824,8.142,149.506
C04393=1121.786,107.843,-57.500,-179.827,8.138,149.506
C04394=1121.790,107.594,-57.481,-179.829,8.134,149.506
C04395=1121.795,107.345,-57.461,-179.831,8.131,149.505
C04396=1121.801,107.096,-57.442,-179.834,8.127,149.505
C04397=1121.805,106.847,-57.423,-179.836,8.123,149.505
C04398=1121.810,106.598,-57.404,-179.838,8.118,149.504
C04399=1121.815,106.348,-57.384,-179.840,8.115,149.504
C04400=1121.819,106.100,-57.365,-179.842,8.111,149.504
C04401=1121.824,105.849,-57.346,-179.845,8.107,149.504
C04402=1121.829,105.600,-57.327,-179.846,8.103,149.503
C04403=1121.834,105.351,-57.308,-179.848,8.100,149.503
C04404=1121.838,105.102,-57.288,-179.850,8.096,149.503
C04405=1121.844,104.853,-57.269,-179.853,8.092,149.502
C04406=1121.848,104.604,-57.250,-179.855,8.088,149.502
C04407=1121.853,104.354,-57.231,-179.857,8.084,149.502
C04408=1121.857,104.105,-57.212,-179.859,8.080,149.502
C04409=1121.862,103.890,-57.196,-179.860,8.077,149.501
C04410=1121.867,103.676,-57.179,-179.862,8.074,149.501
C04411=1121.870,103.462,-57.163,-179.864,8.070,149.501
C04412=1121.875,103.247,-57.146,-179.865,8.067,149.500
C04413=1121.879,103.033,-57.130,-179.867,8.063,149.500
C04414=1121.883,102.818,-57.114,-179.870,8.060,149.500
C04415=1121.887,102.603,-57.098,-179.871,8.057,149.500
C04416=1121.891,102.389,-57.081,-179.873,8.053,149.499
C04417=1121.896,102.141,-57.062,-179.874,8.049,149.499
C04418=1121.901,101.891,-57.043,-179.876,8.046,149.499
C04419=1121.906,101.642,-57.025,-179.878,8.041,149.498
C04420=1121.910,101.392,-57.005,-179.881,8.038,149.498
C04421=1121.915,101.143,-56.987,-179.882,8.034,149.498
C04422=1121.920,100.893,-56.967,-179.884,8.030,149.497
C04423=1121.925,100.645,-56.949,-179.886,8.027,149.497
C04424=1121.930,100.395,-56.930,-179.888,8.022,149.497
C04425=1121.934,100.146,-56.911,-179.890,8.018,149.496
C04426=1121.940,99.897,-56.892,-179.892,8.014,149.496
C04427=1121.944,99.647,-56.873,-179.893,8.011,149.495
C04428=1121.949,99.399,-56.855,-179.895,8.007,149.495
C04429=1121.954,99.149,-56.836,-179.897,8.003,149.495
C04430=1121.958,98.900,-56.817,-179.899,7.999,149.494
C04431=1121.964,98.651,-56.798,-179.901,7.995,149.494
C04432=1121.968,98.401,-56.779,-179.903,7.991,149.494
C04433=1121.973,98.152,-56.761,-179.904,7.987,149.493
C04434=1121.978,97.903,-56.742,-179.906,7.983,149.493
C04435=1121.982,97.653,-56.724,-179.908,7.979,149.492
C04436=1121.988,97.405,-56.704,-179.909,7.976,149.492
C04437=1121.993,97.155,-56.686,-179.911,7.972,149.492
C04438=1121.997,96.906,-56.668,-179.914,7.967,149.491
C04439=1122.002,96.657,-56.649,-179.915,7.964,149.491
C04440=1122.007,96.407,-56.631,-179.917,7.960,149.491
C04441=1122.011,96.158,-56.612,-179.918,7.956,149.490
C04442=1122.017,95.909,-56.593,-179.920,7.952,149.490
C04443=1122.022,95.660,-56.575,-179.922,7.948,149.489
C04444=1122.026,95.410,-56.556,-179.923,7.944,149.489
C04445=1122.031,95.161,-56.538,-179.925,7.940,149.488
C04446=1122.036,94.912,-56.519,-179.926,7.936,149.488
C04447=1122.040,94.662,-56.501,-179.928,7.933,149.488
C04448=1122.045,94.413,-56.483,-179.930,7.929,149.487
C04449=1122.051,94.164,-56.464,-179.932,7.925,149.487
C04450=1122.056,93.915,-56.445,-179.933,7.921,149.486
C04451=1122.060,93.665,-56.427,-179.935,7.917,149.486
C04452=1122.065,93.416,-56.409,-179.936,7.913,149.486
C04453=1122.070,93.167,-56.390,-179.938,7.909,149.485
C04454=1122.075,92.918,-56.372,-179.939,7.905,149.485
C04455=1122.079,92.668,-56.353,-179.941,7.901,149.484
C04456=1122.084,92.419,-56.335,-179.942,7.897,149.484
C04457=1122.090,92.170,-56.316,-179.944,7.894,149.483
C04458=1122.095,91.921,-56.298,-179.945,7.890,149.483
C04459=1122.099,91.671,-56.280,-179.947,7.886,149.482
C04460=1122.104,91.422,-56.262,-179.949,7.882,149.482
C04461=1122.109,91.173,-56.244,-179.950,7.878,149.482
C04462=1122.114,90.923,-56.225,-179.952,7.874,149.481
C04463=1122.118,90.674,-56.206,-179.953,7.870,149.481
C04464=1122.123,90.425,-56.188,-179.954,7.867,149.480
C04465=1122.127,90.210,-56.173,-179.956,7.863,149.480
C04466=1122.131,89.995,-56.157,-179.957,7.860,149.479
C04467=1122.135,89.781,-56.141,-179.959,7.856,149.479
C04468=1122.139,89.567,-56.126,-179.960,7.853,149.478
C04469=1122.144,89.352,-56.110,-179.961,7.850,149.478
C04470=1122.148,89.137,-56.095,-179.962,7.846,149.478
C04471=1122.153,88.923,-56.079,-179.963,7.843,149.477
C04472=1122.157,88.709,-56.063,-179.964,7.840,149.477
C04473=1122.161,88.459,-56.045,-179.966,7.836,149.476
C04474=1122.166,88.210,-56.027,-179.967,7.832,149.476
C04475=1122.171,87.960,-56.009,-179.969,7.828,149.475
C04476=1122.176,87.711,-55.991,-179.969,7.825,149.475
C04477=1122.181,87.462,-55.973,-179.971,7.821,149.474
C04478=1122.187,87.213,-55.955,-179.973,7.817,149.474
C04479=1122.191,86.963,-55.937,-179.974,7.813,149.473
C04480=1122.196,86.714,-55.918,-179.975,7.809,149.473
C04481=1122.201,86.464,-55.900,-179.976,7.806,149.472
C04482=1122.206,86.215,-55.882,-179.978,7.802,149.472
C04483=1122.211,85.966,-55.864,-179.979,7.797,149.471
C04484=1122.215,85.717,-55.846,-179.981,7.793,149.471
C04485=1122.220,85.468,-55.828,-179.982,7.790,149.471
C04486=1122.225,85.218,-55.810,-179.983,7.786,149.470
C04487=1122.230,84.969,-55.792,-179.984,7.782,149.469
C04488=1122.234,84.719,-55.774,-179.985,7.778,149.469
C04489=1122.240,84.470,-55.757,-179.986,7.775,149.468
C04490=1122.245,84.220,-55.739,-179.988,7.771,149.468
C04491=1122.250,83.971,-55.721,-179.989,7.767,149.467
C04492=1122.254,83.722,-55.703,-179.990,7.764,149.467
C04493=1122.259,83.473,-55.685,-179.991,7.759,149.466
C04494=1122.264,83.224,-55.668,-179.993,7.755,149.466
C04495=1122.269,82.974,-55.650,-179.994,7.752,149.465
C04496=1122.274,82.725,-55.632,-179.995,7.748,149.465
C04497=1122.279,82.476,-55.614,-179.996,7.744,149.464
C04498=1122.283,82.227,-55.596,-179.997,7.741,149.464
C04499=1122.288,81.978,-55.578,-179.999,7.737,149.463
C04500=1122.294,81.728,-55.561,-179.999,7.733,149.463
C04501=1122.299,81.479,-55.543,179.999,7.729,149.462
C04502=1122.303,81.229,-55.525,179.998,7.725,149.462
C04503=1122.308,80.980,-55.507,179.997,7.722,149.461
C04504=1122.313,80.730,-55.489,179.996,7.718,149.460
C04505=1122.317,80.481,-55.472,179.995,7.714,149.460
C04506=1122.322,80.232,-55.454,179.994,7.710,149.459
C04507=1122.327,79.983,-55.436,179.993,7.707,149.459
C04508=1122.332,79.733,-55.419,179.992,7.703,149.458
C04509=1122.337,79.484,-55.401,179.991,7.700,149.458
C04510=1122.342,79.234,-55.383,179.990,7.695,149.457
C04511=1122.347,78.985,-55.366,179.989,7.692,149.457
C04512=1122.351,78.736,-55.348,179.988,7.688,149.456
C04513=1122.356,78.487,-55.330,179.987,7.685,149.456
C04514=1122.362,78.237,-55.313,179.986,7.681,149.455
C04515=1122.366,77.988,-55.295,179.985,7.677,149.455
C04516=1122.371,77.738,-55.277,179.984,7.673,149.454
C04517=1122.376,77.489,-55.260,179.983,7.670,149.453
C04518=1122.381,77.240,-55.242,179.982,7.666,149.453
C04519=1122.386,76.990,-55.225,179.981,7.662,149.452
C04520=1122.391,76.741,-55.208,179.979,7.658,149.452
C04521=1122.396,76.527,-55.192,179.978,7.655,149.451
C04522=1122.400,76.312,-55.177,179.978,7.652,149.451
C04523=1122.403,76.097,-55.163,179.976,7.648,149.451
C04524=1122.408,75.882,-55.147,179.975,7.645,149.450
C04525=1122.412,75.668,-55.132,179.973,7.641,149.450
C04526=1122.416,75.454,-55.117,179.972,7.638,149.449
C04527=1122.421,75.238,-55.102,179.971,7.635,149.449
C04528=1122.425,75.023,-55.087,179.970,7.631,149.448
C04529=1122.429,74.775,-55.069,179.968,7.627,149.448
C04530=1122.434,74.525,-55.052,179.967,7.623,149.448
C04531=1122.440,74.276,-55.035,179.966,7.619,149.447
C04532=1122.444,74.027,-55.018,179.964,7.615,149.447
C04533=1122.449,73.778,-55.000,179.962,7.611,149.446
C04534=1122.454,73.528,-54.983,179.961,7.607,149.446
C04535=1122.459,73.279,-54.965,179.960,7.603,149.445
C04536=1122.464,73.029,-54.948,179.958,7.599,149.445
C04537=1122.469,72.779,-54.931,179.957,7.596,149.444
C04538=1122.473,72.531,-54.913,179.956,7.592,149.444
C04539=1122.478,72.281,-54.896,179.955,7.588,149.443
C04540=1122.484,72.032,-54.879,179.953,7.584,149.443
C04541=1122.488,71.783,-54.862,179.951,7.580,149.442
C04542=1122.494,71.533,-54.845,179.950,7.576,149.442
C04543=1122.499,71.284,-54.827,179.949,7.572,149.441
C04544=1122.503,71.034,-54.810,179.947,7.568,149.441
C04545=1122.508,70.785,-54.793,179.946,7.564,149.440
C04546=1122.512,70.536,-54.775,179.944,7.560,149.440
C04547=1122.518,70.287,-54.758,179.943,7.556,149.439
C04548=1122.523,70.037,-54.742,179.941,7.552,149.439
C04549=1122.528,69.787,-54.724,179.940,7.548,149.438
C04550=1122.533,69.538,-54.706,179.939,7.544,149.438
C04551=1122.537,69.289,-54.690,179.937,7.540,149.437
C04552=1122.543,69.040,-54.673,179.935,7.536,149.437
C04553=1122.548,68.790,-54.656,179.934,7.532,149.436
C04554=1122.553,68.541,-54.638,179.933,7.528,149.436
C04555=1122.557,68.291,-54.622,179.932,7.525,149.435
C04556=1122.562,68.042,-54.604,179.931,7.520,149.435
C04557=1122.567,67.793,-54.588,179.929,7.516,149.434
C04558=1122.572,67.544,-54.570,179.928,7.513,149.434
C04559=1122.577,67.294,-54.553,179.926,7.508,149.433
C04560=1122.582,67.044,-54.536,179.925,7.504,149.433
C04561=1122.586,66.795,-54.519,179.923,7.500,149.432
C04562=1122.592,66.546,-54.503,179.922,7.497,149.432
C04563=1122.597,66.296,-54.486,179.921,7.492,149.431
C04564=1122.602,66.047,-54.469,179.919,7.488,149.431
C04565=1122.606,65.798,-54.451,179.918,7.484,149.430
C04566=1122.611,65.549,-54.435,179.916,7.480,149.430
C04567=1122.616,65.299,-54.418,179.915,7.476,149.429
C04568=1122.621,65.050,-54.401,179.913,7.472,149.429
C04569=1122.626,64.800,-54.384,179.912,7.468,149.428
C04570=1122.631,64.551,-54.367,179.911,7.464,149.428
C04571=1122.636,64.301,-54.350,179.909,7.460,149.427
C04572=1122.641,64.052,-54.333,179.909,7.457,149.427
C04573=1122.646,63.803,-54.317,179.907,7.453,149.426
C04574=1122.651,63.553,-54.300,179.906,7.448,149.426
C04575=1122.656,63.304,-54.283,179.904,7.445,149.425
C04576=1122.660,63.054,-54.267,179.903,7.441,149.425
C04577=1122.665,62.840,-54.252,179.901,7.437,149.424
C04578=1122.669,62.625,-54.237,179.900,7.434,149.424
C04579=1122.674,62.410,-54.223,179.899,7.431,149.424
C04580=1122.677,62.195,-54.209,179.898,7.427,149.423
C04581=1122.682,61.981,-54.195,179.897,7.423,149.423
C04582=1122.686,61.766,-54.181,179.896,7.419,149.422
C04583=1122.690,61.551,-54.165,179.895,7.416,149.422
C04584=1122.694,61.337,-54.152,179.894,7.413,149.421
C04585=1122.700,61.087,-54.134,179.892,7.409,149.421
C04586=1122.705,60.838,-54.118,179.891,7.405,149.420
C04587=1122.709,60.589,-54.101,179.890,7.401,149.420
C04588=1122.715,60.338,-54.085,179.888,7.397,149.419
C04589=1122.720,60.089,-54.069,179.887,7.393,149.419
C04590=1122.724,59.840,-54.052,179.885,7.389,149.418
C04591=1122.729,59.590,-54.035,179.884,7.385,149.418
C04592=1122.735,59.341,-54.018,179.883,7.381,149.417
C04593=1122.739,59.092,-54.002,179.881,7.377,149.417
C04594=1122.745,58.843,-53.986,179.880,7.372,149.416
C04595=1122.749,58.593,-53.969,179.878,7.368,149.416
C04596=1122.754,58.343,-53.952,179.878,7.365,149.415
C04597=1122.759,58.094,-53.936,179.876,7.361,149.415
C04598=1122.764,57.845,-53.919,179.875,7.357,149.414
C04599=1122.769,57.596,-53.904,179.874,7.353,149.413
C04600=1122.774,57.346,-53.887,179.872,7.349,149.413
C04601=1122.779,57.096,-53.870,179.871,7.345,149.412
C04602=1122.784,56.847,-53.853,179.870,7.341,149.412
C04603=1122.789,56.597,-53.837,179.868,7.336,149.411
C04604=1122.794,56.349,-53.821,179.867,7.332,149.411
C04605=1122.798,56.099,-53.804,179.865,7.329,149.410
C04606=1122.804,55.850,-53.789,179.864,7.324,149.410
C04607=1122.809,55.600,-53.772,179.863,7.320,149.409
C04608=1122.814,55.351,-53.755,179.862,7.316,149.409
C04609=1122.819,55.101,-53.739,179.860,7.312,149.408
C04610=1122.824,54.852,-53.723,179.859,7.308,149.408
C04611=1122.828,54.603,-53.706,179.858,7.305,149.407
C04612=1122.834,54.353,-53.691,179.857,7.300,149.407
C04613=1122.838,54.104,-53.674,179.855,7.297,149.406
C04614=1122.843,53.854,-53.658,179.854,7.292,149.405
C04615=1122.849,53.605,-53.641,179.853,7.288,149.405
C04616=1122.854,53.355,-53.625,179.852,7.284,149.404
C04617=1122.859,53.106,-53.609,179.850,7.280,149.404
C04618=1122.864,52.857,-53.593,179.849,7.276,149.403
C04619=1122.869,52.607,-53.577,179.847,7.272,149.403
C04620=1122.874,52.358,-53.560,179.846,7.268,149.402
C04621=1122.878,52.108,-53.544,179.845,7.264,149.402
C04622=1122.883,51.859,-53.528,179.844,7.259,149.401
C04623=1122.888,51.609,-53.512,179.842,7.255,149.401
C04624=1122.893,51.360,-53.496,179.841,7.251,149.400
C04625=1122.898,51.110,-53.480,179.839,7.247,149.400
C04626=1122.903,50.861,-53.464,179.839,7.244,149.399
C04627=1122.908,50.611,-53.448,179.838,7.239,149.398
C04628=1122.913,50.362,-53.432,179.836,7.235,149.398
C04629=1122.918,50.112,-53.415,179.835,7.231,149.397
C04630=1122.923,49.863,-53.400,179.834,7.227,149.397
C04631=1122.928,49.614,-53.384,179.833,7.223,149.396
C04632=1122.933,49.364,-53.368,179.831,7.219,149.396
C04633=1122.937,49.150,-53.354,179.830,7.215,149.395
C04634=1122.941,48.935,-53.340,179.829,7.212,149.395
C04635=1122.946,48.720,-53.327,179.828,7.209,149.394
C04636=1122.951,48.505,-53.312,179.827,7.205,149.394
C04637=1122.954,48.290,-53.298,179.826,7.201,149.393
C04638=1122.959,48.075,-53.285,179.825,7.198,149.393
C04639=1122.963,47.860,-53.271,179.824,7.194,149.392
C04640=1122.967,47.646,-53.258,179.823,7.191,149.392
C04641=1122.972,47.396,-53.242,179.822,7.187,149.391
C04642=1122.977,47.146,-53.226,179.820,7.183,149.391
C04643=1122.982,46.898,-53.210,179.819,7.178,149.390
C04644=1122.988,46.648,-53.194,179.818,7.174,149.390
C04645=1122.992,46.398,-53.178,179.816,7.170,149.389
C04646=1122.998,46.149,-53.162,179.815,7.166,149.389
C04647=1123.002,45.900,-53.147,179.814,7.162,149.388
C04648=1123.007,45.650,-53.131,179.813,7.158,149.387
C04649=1123.012,45.401,-53.115,179.812,7.153,149.387
C04650=1123.017,45.151,-53.099,179.810,7.149,149.386
C04651=1123.022,44.902,-53.083,179.809,7.145,149.386
C04652=1123.028,44.652,-53.068,179.808,7.141,149.385
C04653=1123.032,44.403,-53.052,179.806,7.137,149.385
C04654=1123.037,44.153,-53.037,179.806,7.133,149.384
C04655=1123.042,43.904,-53.021,179.805,7.129,149.383
C04656=1123.048,43.655,-53.005,179.803,7.125,149.383
C04657=1123.052,43.405,-52.989,179.802,7.121,149.382
C04658=1123.057,43.156,-52.974,179.801,7.117,149.382
C04659=1123.062,42.906,-52.958,179.800,7.112,149.381
C04660=1123.067,42.656,-52.942,179.798,7.108,149.381
C04661=1123.073,42.407,-52.927,179.797,7.104,149.380
C04662=1123.077,42.158,-52.912,179.796,7.100,149.379
C04663=1123.083,41.908,-52.896,179.795,7.096,149.379
C04664=1123.087,41.658,-52.880,179.794,7.091,149.378
C04665=1123.092,41.410,-52.864,179.793,7.087,149.378
C04666=1123.097,41.160,-52.849,179.792,7.083,149.377
C04667=1123.102,40.910,-52.833,179.790,7.079,149.376
C04668=1123.107,40.661,-52.817,179.789,7.075,149.376
C04669=1123.112,40.412,-52.802,179.788,7.070,149.375
C04670=1123.117,40.162,-52.787,179.787,7.066,149.374
C04671=1123.122,39.912,-52.771,179.785,7.062,149.374
C04672=1123.127,39.663,-52.756,179.784,7.058,149.373
C04673=1123.132,39.414,-52.740,179.783,7.053,149.373
C04674=1123.137,39.164,-52.725,179.782,7.049,149.372
C04675=1123.142,38.915,-52.710,179.780,7.045,149.372
C04676=1123.147,38.665,-52.694,179.779,7.041,149.371
C04677=1123.153,38.415,-52.679,179.778,7.037,149.370
C04678=1123.157,38.166,-52.664,179.778,7.033,149.370
C04679=1123.163,37.917,-52.648,179.777,7.029,149.369
C04680=1123.168,37.667,-52.633,179.776,7.024,149.368
C04681=1123.172,37.418,-52.617,179.774,7.021,149.368
C04682=1123.177,37.168,-52.602,179.773,7.016,149.367
C04683=1123.182,36.919,-52.587,179.772,7.012,149.367
C04684=1123.187,36.670,-52.571,179.771,7.008,149.366
C04685=1123.193,36.420,-52.555,179.770,7.003,149.365
C04686=1123.198,36.171,-52.541,179.769,6.999,149.365
C04687=1123.203,35.920,-52.525,179.767,6.995,149.364
C04688=1123.207,35.671,-52.510,179.766,6.991,149.364
C04689=1123.212,35.456,-52.497,179.765,6.986,149.363
C04690=1123.216,35.241,-52.484,179.764,6.983,149.363
C04691=1123.221,35.027,-52.471,179.764,6.980,149.362
C04692=1123.225,34.812,-52.458,179.762,6.976,149.362
C04693=1123.229,34.596,-52.444,179.762,6.972,149.361
C04694=1123.234,34.382,-52.431,179.760,6.968,149.360
C04695=1123.238,34.167,-52.419,179.760,6.965,149.360
C04696=1123.242,33.952,-52.406,179.758,6.961,149.359
C04697=1123.248,33.703,-52.390,179.757,6.957,149.359
C04698=1123.252,33.453,-52.375,179.756,6.952,149.358
C04699=1123.258,33.204,-52.360,179.755,6.948,149.357
C04700=1123.262,32.954,-52.345,179.754,6.944,149.357
C04701=1123.268,32.704,-52.329,179.753,6.939,149.356
C04702=1123.272,32.455,-52.314,179.752,6.935,149.355
C04703=1123.278,32.205,-52.300,179.751,6.931,149.355
C04704=1123.283,31.956,-52.285,179.750,6.927,149.354
C04705=1123.288,31.707,-52.269,179.749,6.923,149.354
C04706=1123.293,31.457,-52.255,179.748,6.919,149.353
C04707=1123.298,31.208,-52.240,179.747,6.914,149.352
C04708=1123.303,30.958,-52.224,179.746,6.910,149.352
C04709=1123.308,30.709,-52.210,179.745,6.906,149.351
C04710=1123.313,30.459,-52.194,179.744,6.901,149.350
C04711=1123.318,30.210,-52.180,179.743,6.897,149.350
C04712=1123.323,29.961,-52.165,179.742,6.893,149.349
C04713=1123.328,29.711,-52.149,179.741,6.888,149.348
C04714=1123.333,29.461,-52.135,179.740,6.884,149.348
C04715=1123.338,29.211,-52.119,179.739,6.880,149.347
C04716=1123.343,28.962,-52.105,179.738,6.876,149.346
C04717=1123.348,28.712,-52.090,179.737,6.871,149.346
C04718=1123.353,28.462,-52.075,179.736,6.867,149.345
C04719=1123.358,28.213,-52.060,179.734,6.862,149.344
C04720=1123.363,27.964,-52.046,179.733,6.857,149.344
C04721=1123.368,27.714,-52.030,179.732,6.853,149.343
C04722=1123.373,27.465,-52.016,179.731,6.849,149.342
C04723=1123.378,27.215,-52.001,179.730,6.845,149.342
C04724=1123.384,26.965,-51.986,179.729,6.840,149.341
C04725=1123.388,26.716,-51.971,179.728,6.836,149.341
C04726=1123.393,26.467,-51.957,179.727,6.832,149.340
C04727=1123.399,26.218,-51.943,179.726,6.827,149.339
C04728=1123.404,25.968,-51.927,179.725,6.823,149.338
C04729=1123.409,25.719,-51.913,179.724,6.818,149.338
C04730=1123.414,25.469,-51.898,179.723,6.814,149.337
C04731=1123.419,25.219,-51.883,179.722,6.810,149.336
C04732=1123.424,24.970,-51.869,179.721,6.805,149.336
C04733=1123.429,24.721,-51.854,179.720,6.801,149.335
C04734=1123.434,24.471,-51.840,179.719,6.796,149.334
C04735=1123.439,24.222,-51.825,179.718,6.792,149.334
C04736=1123.444,23.972,-51.810,179.717,6.788,149.333
C04737=1123.449,23.722,-51.795,179.716,6.783,149.332
C04738=1123.454,23.472,-51.781,179.715,6.779,149.332
C04739=1123.459,23.223,-51.766,179.714,6.774,149.331
C04740=1123.464,22.974,-51.752,179.713,6.770,149.330
C04741=1123.470,22.724,-51.737,179.712,6.766,149.329
C04742=1123.475,22.475,-51.722,179.711,6.761,149.329
C04743=1123.480,22.225,-51.708,179.710,6.757,149.328
C04744=1123.485,21.976,-51.694,179.710,6.752,149.327
C04745=1123.489,21.761,-51.681,179.709,6.748,149.327
C04746=1123.494,21.546,-51.669,179.708,6.745,149.326
C04747=1123.498,21.331,-51.656,179.707,6.741,149.326
C04748=1123.502,21.116,-51.644,179.706,6.737,149.325
C04749=1123.507,20.900,-51.631,179.705,6.733,149.324
C04750=1123.511,20.686,-51.619,179.705,6.729,149.324
C04751=1123.515,20.471,-51.606,179.703,6.725,149.323
C04752=1123.520,20.255,-51.594,179.703,6.722,149.323
C04753=1123.525,20.005,-51.580,179.702,6.717,149.322
C04754=1123.530,19.756,-51.565,179.701,6.713,149.321
C04755=1123.535,19.507,-51.550,179.700,6.708,149.320
C04756=1123.540,19.257,-51.536,179.700,6.704,149.319
C04757=1123.545,19.008,-51.522,179.698,6.699,149.319
C04758=1123.550,18.758,-51.508,179.697,6.695,149.318
C04759=1123.555,18.509,-51.494,179.696,6.689,149.317
C04760=1123.560,18.259,-51.479,179.695,6.685,149.317
C04761=1123.565,18.009,-51.465,179.694,6.681,149.316
C04762=1123.571,17.760,-51.451,179.694,6.676,149.315
C04763=1123.575,17.511,-51.436,179.693,6.672,149.314
C04764=1123.580,17.261,-51.422,179.692,6.667,149.314
C04765=1123.585,17.012,-51.408,179.691,6.663,149.313
C04766=1123.590,16.762,-51.393,179.690,6.658,149.312
C04767=1123.596,16.513,-51.379,179.689,6.654,149.311
C04768=1123.601,16.263,-51.365,179.688,6.649,149.311
C04769=1123.606,16.013,-51.351,179.688,6.645,149.310
C04770=1123.611,15.764,-51.336,179.687,6.640,149.309
C04771=1123.616,15.514,-51.322,179.685,6.635,149.309
C04772=1123.621,15.265,-51.308,179.685,6.631,149.308
C04773=1123.626,15.015,-51.294,179.684,6.626,149.307
C04774=1123.631,14.766,-51.280,179.683,6.622,149.306
C04775=1123.636,14.516,-51.265,179.682,6.617,149.306
C04776=1123.642,14.266,-51.252,179.681,6.612,149.305
C04777=1123.647,14.017,-51.238,179.680,6.608,149.304
C04778=1123.652,13.767,-51.224,179.680,6.603,149.303
C04779=1123.657,13.518,-51.210,179.679,6.599,149.302
C04780=1123.662,13.268,-51.196,179.678,6.594,149.302
C04781=1123.667,13.018,-51.181,179.677,6.589,149.301
C04782=1123.671,12.769,-51.168,179.676,6.585,149.300
C04783=1123.677,12.520,-51.154,179.675,6.580,149.299
C04784=1123.682,12.270,-51.139,179.674,6.576,149.299
C04785=1123.687,12.020,-51.126,179.674,6.571,149.298
C04786=1123.693,11.771,-51.112,179.673,6.567,149.297
C04787=1123.698,11.521,-51.098,179.672,6.562,149.296
C04788=1123.703,11.272,-51.083,179.671,6.557,149.295
C04789=1123.708,11.023,-51.070,179.671,6.553,149.295
C04790=1123.713,10.772,-51.056,179.670,6.547,149.294
C04791=1123.718,10.523,-51.042,179.669,6.543,149.293
C04792=1123.723,10.274,-51.028,179.668,6.538,149.292
C04793=1123.728,10.024,-51.014,179.667,6.534,149.292
C04794=1123.734,9.774,-51.000,179.666,6.529,149.291
C04795=1123.738,9.525,-50.987,179.666,6.524,149.290
C04796=1123.743,9.275,-50.973,179.665,6.520,149.289
C04797=1123.748,9.026,-50.959,179.664,6.515,149.288
C04798=1123.754,8.776,-50.945,179.663,6.510,149.287
C04799=1123.759,8.526,-50.931,179.662,6.506,149.287
C04800=1123.764,8.278,-50.918,179.662,6.501,149.286
C04801=1123.769,8.062,-50.906,179.662,6.497,149.285
C04802=1123.773,7.847,-50.894,179.661,6.493,149.284
C04803=1123.777,7.631,-50.882,179.660,6.489,149.284
C04804=1123.781,7.416,-50.870,179.660,6.485,149.283
C04805=1123.785,7.201,-50.859,179.660,6.482,149.282
C04806=1123.791,6.986,-50.847,179.659,6.477,149.281
C04807=1123.795,6.771,-50.834,179.659,6.473,149.281
C04808=1123.799,6.556,-50.823,179.658,6.470,149.280
C04809=1123.804,6.306,-50.809,179.658,6.465,149.279
C04810=1123.809,6.057,-50.796,179.657,6.460,149.278
C04811=1123.814,5.807,-50.782,179.657,6.456,149.277
C04812=1123.820,5.558,-50.768,179.657,6.452,149.276
C04813=1123.825,5.308,-50.754,179.656,6.447,149.275
C04814=1123.830,5.059,-50.742,179.655,6.443,149.275
C04815=1123.835,4.809,-50.727,179.655,6.438,149.274
C04816=1123.840,4.559,-50.714,179.655,6.434,149.273
C04817=1123.845,4.310,-50.700,179.654,6.429,149.272
C04818=1123.850,4.060,-50.687,179.654,6.425,149.271
C04819=1123.856,3.811,-50.673,179.653,6.420,149.270
C04820=1123.860,3.561,-50.660,179.652,6.416,149.270
C04821=1123.866,3.312,-50.646,179.652,6.411,149.269
C04822=1123.870,3.062,-50.633,179.652,6.407,149.268
C04823=1123.876,2.813,-50.619,179.651,6.402,149.267
C04824=1123.881,2.562,-50.606,179.651,6.397,149.266
C04825=1123.886,2.314,-50.592,179.650,6.393,149.265
C04826=1123.891,2.063,-50.579,179.649,6.388,149.265
C04827=1123.897,1.814,-50.565,179.649,6.384,149.264
C04828=1123.901,1.564,-50.552,179.649,6.380,149.263
C04829=1123.907,1.315,-50.538,179.648,6.375,149.262
C04830=1123.911,1.065,-50.525,179.647,6.371,149.261
C04831=1123.917,0.816,-50.512,179.647,6.366,149.260
C04832=1123.922,0.566,-50.498,179.646,6.361,149.260
C04833=1123.927,0.317,-50.485,179.646,6.357,149.259
C04834=1123.932,0.067,-50.471,179.645,6.353,149.258
C04835=1123.938,-0.182,-50.458,179.645,6.348,149.257
C04836=1123.943,-0.433,-50.444,179.644,6.344,149.256
C04837=1123.948,-0.681,-50.431,179.644,6.339,149.255
C04838=1123.953,-0.932,-50.418,179.643,6.334,149.255
C04839=1123.958,-1.181,-50.405,179.642,6.330,149.254
C04840=1123.963,-1.431,-50.391,179.642,6.326,149.253
C04841=1123.968,-1.680,-50.378,179.642,6.321,149.252
C04842=1123.974,-1.930,-50.365,179.641,6.317,149.251
C04843=1123.978,-2.179,-50.351,179.640,6.312,149.251
C04844=1123.984,-2.429,-50.338,179.640,6.307,149.250
C04845=1123.989,-2.679,-50.325,179.639,6.303,149.249
C04846=1123.994,-2.928,-50.312,179.638,6.298,149.248
C04847=1123.999,-3.178,-50.298,179.638,6.294,149.247
C04848=1124.004,-3.428,-50.285,179.638,6.290,149.246
C04849=1124.010,-3.677,-50.272,179.637,6.285,149.246
C04850=1124.015,-3.927,-50.259,179.636,6.281,149.245
C04851=1124.020,-4.176,-50.246,179.636,6.276,149.244
C04852=1124.024,-4.426,-50.233,179.635,6.271,149.243
C04853=1124.030,-4.675,-50.219,179.634,6.267,149.242
C04854=1124.035,-4.925,-50.207,179.634,6.262,149.241
C04855=1124.040,-5.175,-50.192,179.633,6.258,149.241
C04856=1124.045,-5.424,-50.180,179.632,6.253,149.240
C04857=1124.050,-5.640,-50.169,179.632,6.249,149.239
C04858=1124.054,-5.855,-50.157,179.631,6.246,149.239
C04859=1124.059,-6.070,-50.146,179.631,6.241,149.238
C04860=1124.063,-6.285,-50.135,179.630,6.238,149.237
C04861=1124.068,-6.500,-50.124,179.629,6.233,149.236
C04862=1124.072,-6.715,-50.112,179.629,6.230,149.236
C04863=1124.077,-6.931,-50.101,179.629,6.226,149.235
C04864=1124.081,-7.146,-50.090,179.628,6.222,149.234
C04865=1124.086,-7.396,-50.077,179.627,6.217,149.234
C04866=1124.091,-7.645,-50.064,179.627,6.212,149.233
C04867=1124.097,-7.895,-50.051,179.626,6.208,149.232
C04868=1124.101,-8.145,-50.038,179.625,6.203,149.231
C04869=1124.106,-8.394,-50.025,179.625,6.199,149.230
C04870=1124.112,-8.644,-50.012,179.624,6.194,149.230
C04871=1124.117,-8.894,-49.999,179.624,6.190,149.229
C04872=1124.122,-9.143,-49.987,179.623,6.186,149.228
C04873=1124.128,-9.393,-49.973,179.622,6.181,149.227
C04874=1124.132,-9.642,-49.960,179.622,6.177,149.226
C04875=1124.137,-9.891,-49.947,179.621,6.172,149.225
C04876=1124.142,-10.141,-49.935,179.620,6.167,149.225
C04877=1124.148,-10.391,-49.921,179.620,6.163,149.224
C04878=1124.153,-10.641,-49.909,179.619,6.158,149.223
C04879=1124.158,-10.890,-49.896,179.618,6.154,149.222
C04880=1124.163,-11.140,-49.884,179.618,6.149,149.221
C04881=1124.169,-11.390,-49.870,179.617,6.144,149.220
C04882=1124.174,-11.639,-49.858,179.616,6.140,149.220
C04883=1124.179,-11.888,-49.845,179.616,6.135,149.219
C04884=1124.184,-12.138,-49.832,179.615,6.130,149.218
C04885=1124.189,-12.388,-49.819,179.614,6.126,149.217
C04886=1124.194,-12.637,-49.806,179.614,6.121,149.216
C04887=1124.199,-12.887,-49.794,179.613,6.116,149.216
C04888=1124.205,-13.136,-49.781,179.612,6.111,149.215
C04889=1124.209,-13.386,-49.768,179.611,6.107,149.214
C04890=1124.215,-13.636,-49.756,179.611,6.102,149.213
C04891=1124.220,-13.886,-49.743,179.610,6.097,149.212
C04892=1124.225,-14.135,-49.730,179.609,6.093,149.212
C04893=1124.230,-14.385,-49.718,179.609,6.088,149.211
C04894=1124.235,-14.634,-49.705,179.608,6.083,149.210
C04895=1124.240,-14.884,-49.692,179.607,6.079,149.209
C04896=1124.246,-15.134,-49.680,179.607,6.074,149.208
C04897=1124.252,-15.383,-49.667,179.606,6.070,149.207
C04898=1124.256,-15.633,-49.654,179.605,6.065,149.207
C04899=1124.261,-15.883,-49.642,179.605,6.061,149.206
C04900=1124.267,-16.132,-49.630,179.604,6.056,149.205
C04901=1124.272,-16.382,-49.617,179.603,6.051,149.204
C04902=1124.277,-16.631,-49.605,179.602,6.046,149.203
C04903=1124.282,-16.880,-49.592,179.602,6.041,149.202
C04904=1124.287,-17.131,-49.580,179.601,6.036,149.202
C04905=1124.292,-17.380,-49.567,179.600,6.032,149.201
C04906=1124.298,-17.630,-49.554,179.600,6.027,149.200
C04907=1124.303,-17.879,-49.541,179.599,6.023,149.199
C04908=1124.308,-18.129,-49.529,179.598,6.018,149.198
C04909=1124.313,-18.379,-49.517,179.597,6.013,149.198
C04910=1124.319,-18.628,-49.504,179.597,6.008,149.197
C04911=1124.323,-18.879,-49.492,179.596,6.003,149.196
C04912=1124.329,-19.128,-49.479,179.595,5.999,149.195
C04913=1124.334,-19.343,-49.469,179.595,5.994,149.194
C04914=1124.337,-19.559,-49.458,179.594,5.991,149.194
C04915=1124.342,-19.774,-49.448,179.593,5.986,149.193
C04916=1124.346,-19.989,-49.437,179.592,5.982,149.192
C04917=1124.351,-20.204,-49.426,179.593,5.978,149.191
C04918=1124.355,-20.420,-49.415,179.592,5.974,149.191
C04919=1124.360,-20.635,-49.405,179.591,5.970,149.190
C04920=1124.365,-20.850,-49.395,179.590,5.966,149.189
C04921=1124.370,-21.099,-49.382,179.590,5.961,149.188
C04922=1124.375,-21.350,-49.370,179.589,5.956,149.188
C04923=1124.380,-21.599,-49.357,179.588,5.951,149.187
C04924=1124.385,-21.849,-49.345,179.587,5.946,149.186
C04925=1124.390,-22.098,-49.333,179.587,5.942,149.185
C04926=1124.396,-22.348,-49.321,179.586,5.937,149.184
C04927=1124.401,-22.598,-49.308,179.585,5.931,149.183
C04928=1124.406,-22.848,-49.296,179.585,5.927,149.182
C04929=1124.411,-23.097,-49.284,179.584,5.922,149.182
C04930=1124.416,-23.347,-49.272,179.583,5.918,149.181
C04931=1124.421,-23.596,-49.260,179.582,5.912,149.180
C04932=1124.427,-23.846,-49.248,179.582,5.907,149.179
C04933=1124.432,-24.096,-49.236,179.581,5.903,149.178
C04934=1124.437,-24.345,-49.223,179.580,5.897,149.177
C04935=1124.443,-24.595,-49.212,179.579,5.893,149.177
C04936=1124.448,-24.844,-49.199,179.579,5.888,149.176
C04937=1124.453,-25.094,-49.187,179.578,5.882,149.175
C04938=1124.458,-25.344,-49.176,179.577,5.878,149.174
C04939=1124.463,-25.593,-49.163,179.577,5.873,149.173
C04940=1124.469,-25.843,-49.151,179.576,5.867,149.172
C04941=1124.474,-26.093,-49.139,179.576,5.863,149.171
C04942=1124.479,-26.342,-49.127,179.577,5.860,149.170
C04943=1124.485,-26.592,-49.115,179.578,5.856,149.169
C04944=1124.489,-26.842,-49.104,179.578,5.851,149.168
C04945=1124.494,-27.091,-49.091,179.579,5.848,149.167
C04946=1124.500,-27.341,-49.079,179.580,5.843,149.166
C04947=1124.505,-27.591,-49.067,179.581,5.840,149.165
C04948=1124.510,-27.840,-49.055,179.582,5.836,149.163
C04949=1124.515,-28.090,-49.043,179.582,5.831,149.162
C04950=1124.521,-28.340,-49.031,179.583,5.827,149.161
C04951=1124.526,-28.589,-49.019,179.583,5.823,149.160
C04952=1124.531,-28.839,-49.007,179.584,5.819,149.159
C04953=1124.536,-29.089,-48.995,179.585,5.815,149.158
C04954=1124.541,-29.338,-48.983,179.585,5.811,149.157
C04955=1124.546,-29.588,-48.971,179.585,5.807,149.156
C04956=1124.552,-29.838,-48.959,179.586,5.803,149.155
C04957=1124.557,-30.088,-48.947,179.586,5.799,149.154
C04958=1124.562,-30.336,-48.936,179.586,5.794,149.153
C04959=1124.568,-30.586,-48.924,179.586,5.790,149.152
C04960=1124.573,-30.836,-48.912,179.586,5.786,149.151
C04961=1124.578,-31.086,-48.900,179.587,5.782,149.150
C04962=1124.583,-31.335,-48.888,179.587,5.778,149.149
C04963=1124.588,-31.585,-48.876,179.586,5.773,149.148
C04964=1124.594,-31.835,-48.864,179.586,5.769,149.148
C04965=1124.599,-32.085,-48.852,179.586,5.765,149.147
C04966=1124.604,-32.334,-48.840,179.586,5.761,149.146
C04967=1124.609,-32.584,-48.829,179.586,5.756,149.145
C04968=1124.614,-32.834,-48.817,179.586,5.752,149.144
C04969=1124.619,-33.049,-48.807,179.586,5.748,149.143
C04970=1124.624,-33.265,-48.797,179.585,5.744,149.142
C04971=1124.628,-33.480,-48.786,179.585,5.740,149.142
C04972=1124.632,-33.695,-48.776,179.585,5.736,149.141
C04973=1124.637,-33.910,-48.766,179.584,5.733,149.140
C04974=1124.641,-34.126,-48.756,179.584,5.729,149.139
C04975=1124.646,-34.341,-48.746,179.584,5.724,149.139
C04976=1124.651,-34.556,-48.736,179.583,5.721,149.138
C04977=1124.655,-34.806,-48.724,179.582,5.716,149.137
C04978=1124.661,-35.056,-48.712,179.582,5.712,149.136
C04979=1124.666,-35.306,-48.700,179.581,5.707,149.135
C04980=1124.671,-35.556,-48.689,179.581,5.703,149.135
C04981=1124.676,-35.805,-48.677,179.580,5.698,149.134
C04982=1124.682,-36.055,-48.666,179.579,5.692,149.133
C04983=1124.687,-36.304,-48.654,179.578,5.688,149.132
C04984=1124.693,-36.554,-48.643,179.578,5.683,149.131
C04985=1124.697,-36.803,-48.631,179.576,5.678,149.131
C04986=1124.702,-37.053,-48.619,179.576,5.673,149.130
C04987=1124.708,-37.303,-48.607,179.575,5.669,149.129
C04988=1124.713,-37.552,-48.596,179.574,5.663,149.128
C04989=1124.718,-37.802,-48.584,179.573,5.659,149.128
C04990=1124.723,-38.052,-48.573,179.572,5.653,149.127
C04991=1124.729,-38.302,-48.562,179.570,5.648,149.126
C04992=1124.734,-38.552,-48.550,179.569,5.644,149.125
C04993=1124.740,-38.801,-48.539,179.568,5.638,149.124
C04994=1124.745,-39.051,-48.527,179.567,5.633,149.124
C04995=1124.750,-39.301,-48.516,179.565,5.628,149.123
C04996=1124.755,-39.551,-48.504,179.564,5.622,149.122
C04997=1124.760,-39.800,-48.492,179.563,5.617,149.122
C04998=1124.766,-40.049,-48.481,179.561,5.612,149.121
C04999=1124.771,-40.299,-48.470,179.560,5.607,149.120
C05000=1124.776,-40.549,-48.458,179.558,5.601,149.119
C05001=1124.782,-40.798,-48.447,179.557,5.596,149.119
C05002=1124.787,-41.048,-48.436,179.555,5.590,149.118
C05003=1124.792,-41.298,-48.424,179.554,5.585,149.117
C05004=1124.797,-41.548,-48.412,179.552,5.580,149.116
C05005=1124.802,-41.797,-48.402,179.550,5.574,149.116
C05006=1124.807,-42.047,-48.391,179.549,5.568,149.115
C05007=1124.813,-42.297,-48.379,179.547,5.562,149.114
C05008=1124.818,-42.546,-48.368,179.545,5.556,149.114
C05009=1124.824,-42.796,-48.356,179.544,5.551,149.113
C05010=1124.829,-43.046,-48.346,179.542,5.545,149.112
C05011=1124.834,-43.295,-48.335,179.541,5.540,149.111
C05012=1124.839,-43.545,-48.323,179.541,5.535,149.110
C05013=1124.844,-43.795,-48.312,179.542,5.530,149.109
C05014=1124.850,-44.044,-48.301,179.541,5.526,149.108
C05015=1124.855,-44.294,-48.289,179.542,5.521,149.107
C05016=1124.860,-44.544,-48.278,179.542,5.516,149.106
C05017=1124.865,-44.793,-48.268,179.542,5.511,149.104
C05018=1124.871,-45.043,-48.256,179.542,5.507,149.104
C05019=1124.876,-45.294,-48.246,179.542,5.502,149.102
C05020=1124.881,-45.542,-48.235,179.543,5.497,149.101
C05021=1124.887,-45.792,-48.223,179.543,5.493,149.100
C05022=1124.892,-46.043,-48.212,179.543,5.488,149.099
C05023=1124.897,-46.292,-48.201,179.543,5.483,149.098
C05024=1124.902,-46.541,-48.189,179.544,5.478,149.097
C05025=1124.907,-46.757,-48.180,179.544,5.474,149.096
C05026=1124.912,-46.972,-48.171,179.544,5.470,149.095
C05027=1124.916,-47.188,-48.161,179.544,5.466,149.094
C05028=1124.921,-47.403,-48.152,179.544,5.462,149.093
C05029=1124.925,-47.618,-48.142,179.544,5.459,149.092
C05030=1124.929,-47.835,-48.133,179.545,5.455,149.091
C05031=1124.934,-48.050,-48.123,179.545,5.451,149.091
C05032=1124.938,-48.266,-48.114,179.544,5.446,149.090
C05033=1124.944,-48.514,-48.103,179.545,5.441,149.088
C05034=1124.950,-48.765,-48.092,179.545,5.436,149.087
C05035=1124.954,-49.015,-48.081,179.545,5.432,149.086
C05036=1124.960,-49.264,-48.070,179.545,5.427,149.085
C05037=1124.965,-49.514,-48.059,179.546,5.423,149.084
C05038=1124.970,-49.763,-48.049,179.546,5.418,149.083
C05039=1124.976,-50.013,-48.037,179.546,5.413,149.082
C05040=1124.981,-50.263,-48.027,179.546,5.409,149.081
C05041=1124.986,-50.512,-48.015,179.546,5.404,149.080
C05042=1124.991,-50.763,-48.005,179.547,5.400,149.079
C05043=1124.997,-51.012,-47.993,179.547,5.394,149.078
C05044=1125.002,-51.262,-47.983,179.547,5.389,149.077
C05045=1125.007,-51.511,-47.972,179.547,5.385,149.076
C05046=1125.012,-51.761,-47.961,179.547,5.380,149.075
C05047=1125.018,-52.011,-47.951,179.548,5.376,149.073
C05048=1125.023,-52.261,-47.939,179.547,5.371,149.072
C05049=1125.029,-52.510,-47.929,179.548,5.367,149.071
C05050=1125.033,-52.760,-47.918,179.548,5.362,149.070
C05051=1125.039,-53.010,-47.907,179.549,5.357,149.069
C05052=1125.044,-53.260,-47.897,179.548,5.353,149.068
C05053=1125.049,-53.509,-47.886,179.548,5.347,149.067
C05054=1125.054,-53.759,-47.875,179.549,5.343,149.066
C05055=1125.060,-54.008,-47.864,179.549,5.338,149.065
C05056=1125.065,-54.258,-47.853,179.549,5.334,149.064
C05057=1125.070,-54.509,-47.843,179.549,5.329,149.063
C05058=1125.076,-54.758,-47.832,179.550,5.325,149.062
C05059=1125.081,-55.008,-47.821,179.550,5.320,149.061
C05060=1125.086,-55.257,-47.811,179.550,5.315,149.059
C05061=1125.091,-55.507,-47.800,179.550,5.311,149.058
C05062=1125.097,-55.757,-47.790,179.550,5.305,149.057
C05063=1125.102,-56.007,-47.779,179.551,5.301,149.056
C05064=1125.108,-56.256,-47.767,179.550,5.296,149.055
C05065=1125.113,-56.506,-47.757,179.551,5.292,149.054
C05066=1125.118,-56.756,-47.747,179.551,5.287,149.053
C05067=1125.123,-57.005,-47.736,179.551,5.283,149.052
C05068=1125.128,-57.255,-47.725,179.551,5.278,149.051
C05069=1125.134,-57.505,-47.715,179.552,5.273,149.050
C05070=1125.139,-57.755,-47.704,179.552,5.269,149.049
C05071=1125.144,-58.004,-47.693,179.552,5.263,149.048
C05072=1125.149,-58.254,-47.683,179.553,5.259,149.047
C05073=1125.155,-58.503,-47.673,179.552,5.254,149.046
C05074=1125.160,-58.754,-47.662,179.553,5.250,149.044
C05075=1125.165,-59.003,-47.651,179.552,5.245,149.044
C05076=1125.170,-59.253,-47.641,179.553,5.241,149.042
C05077=1125.176,-59.502,-47.630,179.553,5.236,149.041
C05078=1125.181,-59.752,-47.620,179.553,5.232,149.040
C05079=1125.186,-60.002,-47.609,179.554,5.227,149.039
C05080=1125.192,-60.251,-47.599,179.554,5.222,149.038
C05081=1125.196,-60.467,-47.589,179.553,5.217,149.037
C05082=1125.201,-60.683,-47.581,179.552,5.213,149.037
C05083=1125.206,-60.898,-47.572,179.552,5.208,149.036
C05084=1125.210,-61.113,-47.563,179.551,5.204,149.035
C05085=1125.215,-61.329,-47.554,179.550,5.199,149.034
C05086=1125.219,-61.544,-47.544,179.549,5.194,149.033
C05087=1125.224,-61.761,-47.536,179.548,5.190,149.033
C05088=1125.229,-61.976,-47.526,179.548,5.186,149.032
C05089=1125.233,-62.226,-47.516,179.547,5.180,149.031
C05090=1125.239,-62.475,-47.506,179.546,5.175,149.030
C05091=1125.244,-62.725,-47.496,179.545,5.170,149.029
C05092=1125.249,-62.975,-47.485,179.544,5.164,149.028
C05093=1125.255,-63.224,-47.474,179.543,5.159,149.028
C05094=1125.260,-63.474,-47.464,179.543,5.154,149.027
C05095=1125.265,-63.724,-47.454,179.542,5.148,149.026
C05096=1125.271,-63.974,-47.443,179.541,5.142,149.025
C05097=1125.276,-64.224,-47.433,179.541,5.138,149.024
C05098=1125.281,-64.473,-47.423,179.540,5.132,149.023
C05099=1125.286,-64.723,-47.413,179.540,5.127,149.022
C05100=1125.291,-64.973,-47.403,179.539,5.122,149.021
C05101=1125.297,-65.222,-47.392,179.538,5.116,149.020
C05102=1125.302,-65.472,-47.382,179.537,5.111,149.019
C05103=1125.308,-65.721,-47.372,179.537,5.105,149.018
C05104=1125.313,-65.972,-47.362,179.536,5.101,149.017
C05105=1125.318,-66.222,-47.352,179.535,5.095,149.016
C05106=1125.324,-66.471,-47.342,179.535,5.090,149.015
C05107=1125.329,-66.721,-47.332,179.535,5.084,149.014
C05108=1125.334,-66.971,-47.321,179.534,5.079,149.013
C05109=1125.340,-67.220,-47.311,179.533,5.074,149.012
C05110=1125.345,-67.470,-47.302,179.533,5.068,149.011
C05111=1125.350,-67.720,-47.291,179.532,5.063,149.010
C05112=1125.355,-67.969,-47.281,179.531,5.058,149.009
C05113=1125.361,-68.220,-47.271,179.532,5.053,149.008
C05114=1125.367,-68.469,-47.261,179.531,5.047,149.007
C05115=1125.371,-68.719,-47.251,179.531,5.042,149.006
C05116=1125.377,-68.969,-47.241,179.530,5.036,149.005
C05117=1125.382,-69.218,-47.231,179.530,5.031,149.004
C05118=1125.388,-69.468,-47.221,179.529,5.026,149.003
C05119=1125.392,-69.718,-47.211,179.529,5.021,149.002
C05120=1125.398,-69.968,-47.201,179.528,5.015,149.001
C05121=1125.404,-70.217,-47.191,179.528,5.010,149.000
C05122=1125.409,-70.467,-47.181,179.528,5.005,148.999
C05123=1125.414,-70.717,-47.172,179.527,4.999,148.998
C05124=1125.419,-70.967,-47.161,179.527,4.994,148.997
C05125=1125.424,-71.216,-47.152,179.527,4.988,148.996
C05126=1125.430,-71.466,-47.142,179.526,4.984,148.995
C05127=1125.436,-71.716,-47.132,179.526,4.978,148.994
C05128=1125.441,-71.965,-47.122,179.526,4.972,148.992
C05129=1125.447,-72.215,-47.113,179.526,4.968,148.991
C05130=1125.452,-72.466,-47.102,179.526,4.962,148.990
C05131=1125.456,-72.715,-47.093,179.525,4.957,148.989
C05132=1125.462,-72.965,-47.083,179.525,4.952,148.988
C05133=1125.468,-73.214,-47.073,179.525,4.947,148.987
C05134=1125.473,-73.464,-47.063,179.524,4.941,148.986
C05135=1125.479,-73.714,-47.054,179.524,4.936,148.985
C05136=1125.484,-73.963,-47.044,179.524,4.931,148.984
C05137=1125.489,-74.179,-47.036,179.524,4.926,148.983
C05138=1125.493,-74.395,-47.028,179.524,4.921,148.982
C05139=1125.497,-74.611,-47.018,179.524,4.917,148.981
C05140=1125.502,-74.826,-47.010,179.524,4.912,148.980
C05141=1125.507,-75.042,-47.002,179.523,4.908,148.979
C05142=1125.511,-75.257,-46.993,179.524,4.903,148.978
C05143=1125.516,-75.473,-46.985,179.524,4.899,148.977
C05144=1125.520,-75.689,-46.977,179.523,4.894,148.976
C05145=1125.526,-75.939,-46.967,179.523,4.889,148.975
C05146=1125.531,-76.188,-46.958,179.524,4.883,148.974
C05147=1125.537,-76.438,-46.948,179.523,4.879,148.973
C05148=1125.542,-76.688,-46.938,179.523,4.873,148.972
C05149=1125.547,-76.937,-46.928,179.523,4.868,148.971
C05150=1125.553,-77.187,-46.919,179.523,4.862,148.969
C05151=1125.558,-77.437,-46.909,179.523,4.857,148.968
C05152=1125.564,-77.687,-46.900,179.523,4.852,148.967
C05153=1125.569,-77.937,-46.891,179.523,4.847,148.966
C05154=1125.575,-78.186,-46.881,179.524,4.842,148.965
C05155=1125.580,-78.436,-46.872,179.523,4.837,148.964
C05156=1125.586,-78.686,-46.862,179.523,4.832,148.963
C05157=1125.591,-78.935,-46.853,179.524,4.827,148.961
C05158=1125.596,-79.186,-46.842,179.524,4.821,148.960
C05159=1125.601,-79.435,-46.833,179.524,4.816,148.959
C05160=1125.607,-79.686,-46.824,179.524,4.811,148.958
C05161=1125.612,-79.935,-46.814,179.524,4.806,148.957
C05162=1125.617,-80.185,-46.805,179.524,4.801,148.956
C05163=1125.622,-80.434,-46.795,179.525,4.796,148.954
C05164=1125.628,-80.684,-46.786,179.525,4.791,148.953
C05165=1125.633,-80.934,-46.777,179.525,4.785,148.952
C05166=1125.638,-81.183,-46.767,179.525,4.780,148.951
C05167=1125.644,-81.434,-46.758,179.525,4.775,148.950
C05168=1125.649,-81.684,-46.749,179.525,4.770,148.949
C05169=1125.654,-81.933,-46.739,179.526,4.765,148.947
C05170=1125.660,-82.183,-46.730,179.526,4.760,148.946
C05171=1125.665,-82.433,-46.721,179.526,4.754,148.945
C05172=1125.670,-82.682,-46.711,179.527,4.749,148.944
C05173=1125.676,-82.932,-46.702,179.527,4.744,148.943
C05174=1125.681,-83.182,-46.693,179.527,4.738,148.941
C05175=1125.687,-83.432,-46.682,179.528,4.734,148.940
C05176=1125.692,-83.681,-46.674,179.528,4.729,148.939
C05177=1125.698,-83.931,-46.665,179.528,4.724,148.938
C05178=1125.704,-84.181,-46.655,179.528,4.719,148.937
C05179=1125.709,-84.430,-46.646,179.528,4.713,148.936
C05180=1125.714,-84.680,-46.637,179.529,4.708,148.934
C05181=1125.720,-84.930,-46.627,179.530,4.704,148.933
C05182=1125.725,-85.180,-46.619,179.530,4.698,148.932
C05183=1125.730,-85.429,-46.609,179.530,4.693,148.931
C05184=1125.736,-85.679,-46.599,179.530,4.688,148.929
C05185=1125.741,-85.929,-46.591,179.531,4.684,148.928
C05186=1125.746,-86.179,-46.582,179.531,4.679,148.927
C05187=1125.752,-86.429,-46.572,179.532,4.673,148.926
C05188=1125.757,-86.678,-46.563,179.533,4.669,148.924
C05189=1125.762,-86.928,-46.554,179.533,4.663,148.923
C05190=1125.767,-87.178,-46.545,179.533,4.658,148.922
C05191=1125.773,-87.428,-46.535,179.534,4.654,148.921
C05192=1125.778,-87.678,-46.526,179.535,4.648,148.920
C05193=1125.783,-87.893,-46.519,179.535,4.644,148.919
C05194=1125.787,-88.109,-46.511,179.536,4.640,148.917
C05195=1125.792,-88.325,-46.502,179.536,4.636,148.916
C05196=1125.797,-88.540,-46.495,179.537,4.632,148.915
C05197=1125.801,-88.757,-46.487,179.536,4.627,148.914
C05198=1125.806,-88.972,-46.479,179.537,4.623,148.913
C05199=1125.810,-89.187,-46.472,179.537,4.619,148.912
C05200=1125.815,-89.404,-46.463,179.538,4.614,148.911
C05201=1125.821,-89.653,-46.454,179.539,4.610,148.910
C05202=1125.826,-89.903,-46.445,179.539,4.605,148.909
C05203=1125.831,-90.152,-46.437,179.540,4.600,148.908
C05204=1125.837,-90.403,-46.427,179.541,4.595,148.906
C05205=1125.843,-90.652,-46.418,179.541,4.591,148.905
C05206=1125.848,-90.902,-46.410,179.542,4.585,148.904
C05207=1125.853,-91.152,-46.400,179.542,4.581,148.903
C05208=1125.858,-91.401,-46.391,179.543,4.575,148.901
C05209=1125.864,-91.652,-46.382,179.544,4.571,148.900
C05210=1125.869,-91.901,-46.373,179.545,4.567,148.899
C05211=1125.875,-92.151,-46.364,179.545,4.562,148.898
C05212=1125.880,-92.400,-46.355,179.546,4.557,148.896
C05213=1125.885,-92.650,-46.346,179.547,4.552,148.895
C05214=1125.891,-92.900,-46.337,179.547,4.547,148.894
C05215=1125.896,-93.150,-46.328,179.548,4.543,148.893
C05216=1125.901,-93.400,-46.319,179.549,4.538,148.891
C05217=1125.907,-93.649,-46.311,179.549,4.533,148.890
C05218=1125.912,-93.899,-46.302,179.550,4.529,148.889
C05219=1125.917,-94.149,-46.293,179.551,4.524,148.888
C05220=1125.922,-94.399,-46.284,179.552,4.520,148.886
C05221=1125.928,-94.649,-46.274,179.553,4.514,148.885
C05222=1125.933,-94.899,-46.265,179.553,4.509,148.884
C05223=1125.939,-95.148,-46.257,179.554,4.505,148.883
C05224=1125.944,-95.398,-46.248,179.554,4.500,148.881
C05225=1125.950,-95.648,-46.239,179.553,4.495,148.881
C05226=1125.955,-95.898,-46.230,179.554,4.490,148.879
C05227=1125.960,-96.147,-46.221,179.554,4.485,148.878
C05228=1125.967,-96.397,-46.213,179.555,4.480,148.877
C05229=1125.972,-96.647,-46.204,179.555,4.475,148.876
C05230=1125.977,-96.897,-46.195,179.555,4.470,148.875
C05231=1125.982,-97.147,-46.186,179.555,4.465,148.873
C05232=1125.988,-97.396,-46.178,179.556,4.460,148.872
C05233=1125.993,-97.646,-46.169,179.556,4.455,148.871
C05234=1125.998,-97.896,-46.160,179.557,4.450,148.870
C05235=1126.003,-98.146,-46.151,179.557,4.445,148.869
C05236=1126.009,-98.396,-46.142,179.556,4.440,148.868
C05237=1126.015,-98.645,-46.134,179.557,4.435,148.867
C05238=1126.020,-98.895,-46.125,179.557,4.431,148.865
C05239=1126.025,-99.145,-46.116,179.558,4.425,148.864
C05240=1126.030,-99.395,-46.108,179.558,4.420,148.863
C05241=1126.037,-99.644,-46.098,179.558,4.415,148.862
C05242=1126.042,-99.894,-46.090,179.558,4.410,148.861
C05243=1126.047,-100.145,-46.081,179.559,4.405,148.859
C05244=1126.053,-100.394,-46.073,179.559,4.400,148.858
C05245=1126.058,-100.644,-46.064,179.559,4.396,148.857
C05246=1126.063,-100.894,-46.055,179.559,4.390,148.856
C05247=1126.069,-101.143,-46.046,179.560,4.385,148.855
C05248=1126.075,-101.393,-46.038,179.560,4.380,148.854
C05249=1126.079,-101.609,-46.030,179.560,4.376,148.853
C05250=1126.084,-101.825,-46.023,179.560,4.371,148.852
C05251=1126.088,-102.040,-46.015,179.561,4.367,148.851
C05252=1126.093,-102.257,-46.008,179.561,4.363,148.850
C05253=1126.098,-102.472,-46.001,179.561,4.358,148.849
C05254=1126.102,-102.688,-45.993,179.561,4.354,148.848
C05255=1126.107,-102.904,-45.986,179.562,4.350,148.847
C05256=1126.111,-103.120,-45.978,179.561,4.345,148.846
C05257=1126.117,-103.369,-45.970,179.562,4.340,148.844
C05258=1126.123,-103.620,-45.962,179.562,4.335,148.843
C05259=1126.127,-103.869,-45.953,179.562,4.329,148.842
C05260=1126.133,-104.118,-45.945,179.562,4.324,148.841
C05261=1126.138,-104.368,-45.936,179.563,4.320,148.840
C05262=1126.144,-104.619,-45.928,179.563,4.315,148.839
C05263=1126.149,-104.868,-45.919,179.563,4.310,148.838
C05264=1126.155,-105.118,-45.911,179.563,4.305,148.836
C05265=1126.160,-105.368,-45.902,179.564,4.300,148.835
C05266=1126.166,-105.617,-45.894,179.564,4.294,148.834
C05267=1126.171,-105.868,-45.885,179.564,4.289,148.833
C05268=1126.176,-106.118,-45.877,179.564,4.284,148.832
C05269=1126.181,-106.366,-45.869,179.565,4.279,148.830
C05270=1126.187,-106.617,-45.860,179.564,4.274,148.829
C05271=1126.192,-106.867,-45.852,179.565,4.269,148.828
C05272=1126.198,-107.116,-45.844,179.565,4.264,148.827
C05273=1126.203,-107.366,-45.835,179.565,4.259,148.826
C05274=1126.209,-107.615,-45.826,179.565,4.253,148.825
C05275=1126.214,-107.866,-45.818,179.565,4.248,148.823
C05276=1126.219,-108.115,-45.810,179.566,4.243,148.822
C05277=1126.225,-108.365,-45.802,179.566,4.238,148.821
C05278=1126.230,-108.615,-45.793,179.566,4.233,148.820
C05279=1126.236,-108.865,-45.785,179.566,4.228,148.819
C05280=1126.241,-109.115,-45.776,179.567,4.222,148.817
C05281=1126.247,-109.365,-45.768,179.566,4.218,148.817
C05282=1126.252,-109.614,-45.760,179.567,4.212,148.815
C05283=1126.257,-109.864,-45.752,179.567,4.207,148.814
C05284=1126.263,-110.114,-45.744,179.567,4.202,148.813
C05285=1126.269,-110.364,-45.735,179.567,4.197,148.812
C05286=1126.273,-110.614,-45.727,179.568,4.192,148.811
C05287=1126.279,-110.863,-45.719,179.568,4.187,148.809
C05288=1126.284,-111.113,-45.710,179.568,4.181,148.808
C05289=1126.290,-111.363,-45.703,179.568,4.175,148.807
C05290=1126.296,-111.613,-45.694,179.568,4.170,148.806
C05291=1126.301,-111.862,-45.686,179.568,4.165,148.805
C05292=1126.306,-112.113,-45.678,179.569,4.160,148.803
C05293=1126.312,-112.362,-45.670,179.569,4.155,148.802
C05294=1126.318,-112.612,-45.662,179.569,4.150,148.801
C05295=1126.323,-112.861,-45.654,179.569,4.145,148.800
C05296=1126.328,-113.112,-45.645,179.569,4.140,148.799
C05297=1126.334,-113.362,-45.638,179.569,4.134,148.798
C05298=1126.339,-113.611,-45.629,179.569,4.128,148.796
C05299=1126.345,-113.861,-45.621,179.569,4.123,148.795
C05300=1126.350,-114.111,-45.613,179.570,4.118,148.794
C05301=1126.356,-114.360,-45.605,179.570,4.113,148.793
C05302=1126.361,-114.611,-45.597,179.570,4.108,148.792
C05303=1126.366,-114.860,-45.589,179.570,4.103,148.790
C05304=1126.372,-115.110,-45.580,179.571,4.097,148.789
C05305=1126.378,-115.379,-45.573,179.570,4.091,148.788
C05306=1126.383,-115.649,-45.563,179.571,4.086,148.787
C05307=1126.389,-115.918,-45.555,179.571,4.080,148.785
C05308=1126.396,-116.188,-45.546,179.571,4.075,148.784
C05309=1126.400,-116.437,-45.538,179.571,4.069,148.783
C05310=1126.406,-116.687,-45.530,179.571,4.063,148.782
C05311=1126.412,-116.936,-45.523,179.571,4.058,148.781
C05312=1126.417,-117.187,-45.515,179.572,4.053,148.779
C05313=1126.423,-117.436,-45.506,179.572,4.048,148.778
C05314=1126.427,-117.686,-45.499,179.572,4.042,148.777
C05315=1126.434,-117.936,-45.491,179.572,4.037,148.776
C05316=1126.438,-118.186,-45.483,179.572,4.032,148.775
C05317=1126.444,-118.435,-45.475,179.572,4.026,148.773
C05318=1126.450,-118.685,-45.467,179.572,4.020,148.772
C05319=1126.455,-118.935,-45.459,179.572,4.015,148.771
C05320=1126.461,-119.185,-45.452,179.573,4.010,148.770
C05321=1126.466,-119.435,-45.444,179.573,4.005,148.769
C05322=1126.472,-119.685,-45.436,179.573,3.999,148.767
C05323=1126.476,-119.934,-45.428,179.573,3.994,148.766
C05324=1126.482,-120.184,-45.420,179.573,3.989,148.765
C05325=1126.509,-121.405,-45.380,178.429,6.138,149.570
C05326=1126.518,-121.815,-45.367,178.426,6.137,149.570
C05327=1126.524,-122.064,-45.358,178.424,6.137,149.571
C05328=1126.528,-122.314,-45.351,178.422,6.136,149.571
C05329=1126.533,-122.564,-45.342,178.420,6.136,149.572
C05330=1126.540,-122.814,-45.334,178.418,6.136,149.572
C05331=1126.545,-123.064,-45.325,178.417,6.135,149.573
C05332=1126.550,-123.313,-45.318,178.415,6.134,149.573
C05333=1126.556,-123.564,-45.310,178.413,6.134,149.574
C05334=1126.561,-123.813,-45.301,178.411,6.134,149.574
C05335=1126.566,-124.063,-45.293,178.409,6.134,149.575
C05336=1126.572,-124.312,-45.285,178.407,6.133,149.575
C05337=1126.577,-124.563,-45.277,178.405,6.132,149.576
C05338=1126.582,-124.812,-45.268,178.404,6.132,149.576
C05339=1126.588,-125.062,-45.261,178.402,6.131,149.576
C05340=1126.593,-125.312,-45.252,178.400,6.131,149.577
C05341=1126.599,-125.561,-45.244,178.398,6.131,149.577
C05342=1126.604,-125.812,-45.236,178.396,6.131,149.578
C05343=1126.610,-126.061,-45.228,178.394,6.130,149.578
C05344=1126.615,-126.311,-45.220,178.393,6.130,149.579
C05345=1126.621,-126.561,-45.212,178.391,6.129,149.579
C05346=1126.626,-126.811,-45.203,178.389,6.129,149.580
C05347=1126.632,-127.060,-45.196,178.387,6.128,149.580
C05348=1126.637,-127.311,-45.187,178.385,6.128,149.581
C05349=1126.642,-127.560,-45.180,178.383,6.127,149.581
C05350=1126.648,-127.810,-45.171,178.382,6.127,149.581
C05351=1126.654,-128.060,-45.164,178.380,6.126,149.582
C05352=1126.658,-128.309,-45.155,178.378,6.126,149.582
C05353=1126.664,-128.559,-45.147,178.376,6.126,149.583
C05354=1126.670,-128.810,-45.139,178.374,6.126,149.583
C05355=1126.248,-128.820,-45.184,179.584,3.800,148.721
C05356=1126.244,-128.570,-45.192,179.585,3.806,148.722
C05357=1126.237,-128.319,-45.199,179.584,3.812,148.723
C05358=1126.232,-128.070,-45.206,179.585,3.818,148.725
C05359=1126.227,-127.820,-45.213,179.584,3.823,148.726
C05360=1126.221,-127.570,-45.222,179.584,3.829,148.727
C05361=1126.216,-127.320,-45.229,179.584,3.834,148.728
C05362=1126.210,-127.071,-45.236,179.584,3.840,148.730
C05363=1126.204,-126.821,-45.244,179.584,3.845,148.731
C05364=1126.200,-126.571,-45.251,179.583,3.851,148.732
C05365=1126.194,-126.321,-45.259,179.584,3.857,148.733
C05366=1126.188,-126.072,-45.267,179.583,3.862,148.734
C05367=1126.183,-125.821,-45.273,179.583,3.868,148.736
C05368=1126.177,-125.571,-45.281,179.583,3.873,148.737
C05369=1126.172,-125.322,-45.288,179.583,3.879,148.738
C05370=1126.166,-125.072,-45.296,179.583,3.885,148.740
C05371=1126.161,-124.822,-45.304,179.582,3.890,148.741
C05372=1126.155,-124.572,-45.312,179.583,3.896,148.742
C05373=1126.150,-124.323,-45.319,179.582,3.901,148.743
C05374=1126.145,-124.072,-45.326,179.583,3.907,148.744
C05375=1126.139,-123.823,-45.334,179.582,3.912,148.746
C05376=1126.133,-123.573,-45.341,179.582,3.918,148.747
C05377=1126.128,-123.323,-45.350,179.582,3.924,148.748
C05378=1126.123,-123.074,-45.358,179.582,3.929,148.749
C05379=1126.117,-122.823,-45.366,179.581,3.934,148.751
C05380=1126.112,-122.574,-45.373,179.582,3.940,148.752
C05381=1126.106,-122.324,-45.381,179.581,3.945,148.753
C05382=1126.101,-122.074,-45.388,179.581,3.950,148.754
C05383=1126.095,-121.824,-45.396,179.581,3.956,148.755
C05384=1126.090,-121.575,-45.403,179.581,3.962,148.757
C05385=1126.084,-121.324,-45.412,179.581,3.967,148.758
C05386=1126.079,-121.075,-45.419,179.581,3.973,148.759
C05387=1126.074,-120.824,-45.427,179.581,3.978,148.760
C05388=1126.069,-120.576,-45.435,179.580,3.983,148.761
C05389=1126.063,-120.326,-45.443,179.581,3.989,148.763
C05390=1126.057,-120.075,-45.451,179.581,3.994,148.764
C05391=1126.052,-119.826,-45.458,179.580,3.999,148.765
C05392=1126.046,-119.575,-45.466,179.580,4.005,148.766
C05393=1126.041,-119.326,-45.474,179.580,4.011,148.768
C05394=1126.036,-119.076,-45.482,179.579,4.016,148.769
C05395=1126.030,-118.827,-45.490,179.579,4.021,148.770
C05396=1126.024,-118.577,-45.498,179.579,4.027,148.771
C05397=1126.019,-118.326,-45.506,179.579,4.033,148.773
C05398=1126.014,-118.078,-45.514,179.579,4.038,148.774
C05399=1126.008,-117.827,-45.522,179.579,4.043,148.775
C05400=1126.002,-117.577,-45.530,179.578,4.048,148.776
C05401=1125.998,-117.327,-45.537,179.579,4.054,148.777
C05402=1125.992,-117.078,-45.546,179.578,4.059,148.779
C05403=1125.987,-116.828,-45.553,179.578,4.064,148.780
C05404=1125.982,-116.612,-45.560,179.578,4.069,148.781
C05405=1125.977,-116.396,-45.567,179.578,4.073,148.782
C05406=1125.972,-116.180,-45.574,179.578,4.078,148.783
C05407=1125.968,-115.965,-45.581,179.577,4.082,148.784
C05408=1125.963,-115.749,-45.588,179.578,4.087,148.785
C05409=1125.958,-115.532,-45.595,179.578,4.092,148.786
C05410=1125.953,-115.317,-45.602,179.577,4.096,148.787
C05411=1125.949,-115.100,-45.609,179.577,4.101,148.788
C05412=1125.944,-114.851,-45.617,179.577,4.106,148.789
C05413=1125.938,-114.601,-45.625,179.577,4.111,148.790
C05414=1125.932,-114.351,-45.633,179.577,4.117,148.792
C05415=1125.928,-114.102,-45.641,179.576,4.122,148.793
C05416=1125.922,-113.852,-45.649,179.577,4.128,148.794
C05417=1125.916,-113.601,-45.657,179.576,4.133,148.795
C05418=1125.910,-113.352,-45.666,179.576,4.138,148.796
C05419=1125.906,-113.102,-45.673,179.576,4.143,148.798
C05420=1125.900,-112.853,-45.682,179.576,4.149,148.799
C05421=1125.894,-112.602,-45.690,179.576,4.153,148.800
C05422=1125.889,-112.353,-45.697,179.576,4.158,148.801
C05423=1125.884,-112.103,-45.706,179.575,4.164,148.802
C05424=1125.878,-111.853,-45.714,179.575,4.169,148.803
C05425=1125.873,-111.604,-45.723,179.575,4.175,148.804
C05426=1125.867,-111.354,-45.731,179.575,4.180,148.806
C05427=1125.862,-111.104,-45.739,179.575,4.185,148.807
C05428=1125.857,-110.854,-45.747,179.575,4.190,148.808
C05429=1125.851,-110.605,-45.756,179.574,4.196,148.809
C05430=1125.845,-110.354,-45.764,179.574,4.201,148.810
C05431=1125.840,-110.105,-45.773,179.574,4.206,148.812
C05432=1125.835,-109.855,-45.780,179.574,4.211,148.813
C05433=1125.830,-109.605,-45.789,179.573,4.216,148.814
C05434=1125.824,-109.355,-45.797,179.573,4.221,148.815
C05435=1125.818,-109.105,-45.806,179.573,4.227,148.816
C05436=1125.812,-108.856,-45.814,179.573,4.231,148.817
C05437=1125.808,-108.606,-45.822,179.573,4.237,148.819
C05438=1125.802,-108.356,-45.830,179.573,4.242,148.820
C05439=1125.797,-108.106,-45.839,179.572,4.247,148.821
C05440=1125.792,-107.857,-45.847,179.572,4.252,148.822
C05441=1125.785,-107.607,-45.855,179.572,4.257,148.823
C05442=1125.780,-107.357,-45.864,179.572,4.262,148.825
C05443=1125.775,-107.106,-45.872,179.571,4.268,148.826
C05444=1125.770,-106.858,-45.880,179.571,4.273,148.827
C05445=1125.765,-106.608,-45.889,179.571,4.278,148.828
C05446=1125.759,-106.357,-45.897,179.571,4.283,148.829
C05447=1125.753,-106.108,-45.906,179.571,4.288,148.830
C05448=1125.748,-105.858,-45.915,179.571,4.293,148.831
C05449=1125.743,-105.608,-45.923,179.570,4.298,148.833
C05450=1125.737,-105.359,-45.931,179.570,4.303,148.834
C05451=1125.732,-105.109,-45.940,179.570,4.309,148.835
C05452=1125.726,-104.858,-45.949,179.570,4.314,148.836
C05453=1125.721,-104.609,-45.957,179.570,4.319,148.837
C05454=1125.715,-104.359,-45.966,179.569,4.324,148.839
C05455=1125.711,-104.109,-45.974,179.569,4.329,148.840
C05456=1125.705,-103.860,-45.982,179.568,4.334,148.841
C05457=1125.700,-103.610,-45.991,179.569,4.338,148.842
C05458=1125.694,-103.360,-45.999,179.568,4.344,148.843
C05459=1125.689,-103.111,-46.008,179.568,4.349,148.844
C05460=1125.684,-102.895,-46.016,179.568,4.354,148.845
C05461=1125.680,-102.678,-46.023,179.568,4.358,148.847
C05462=1125.675,-102.463,-46.031,179.567,4.362,148.847
C05463=1125.670,-102.247,-46.038,179.568,4.367,148.848
C05464=1125.666,-102.032,-46.045,179.567,4.371,148.849
C05465=1125.661,-101.815,-46.053,179.566,4.375,148.851
C05466=1125.656,-101.600,-46.060,179.567,4.380,148.851
C05467=1125.652,-101.384,-46.068,179.566,4.384,148.852
C05468=1125.646,-101.135,-46.076,179.566,4.389,148.854
C05469=1125.641,-100.885,-46.085,179.566,4.394,148.855
C05470=1125.636,-100.635,-46.094,179.566,4.399,148.856
C05471=1125.630,-100.384,-46.102,179.565,4.404,148.857
C05472=1125.624,-100.135,-46.111,179.565,4.409,148.858
C05473=1125.619,-99.885,-46.120,179.565,4.414,148.859
C05474=1125.613,-99.635,-46.129,179.565,4.419,148.861
C05475=1125.608,-99.385,-46.138,179.565,4.424,148.862
C05476=1125.602,-99.136,-46.146,179.564,4.429,148.863
C05477=1125.597,-98.886,-46.155,179.564,4.434,148.864
C05478=1125.592,-98.636,-46.164,179.563,4.439,148.865
C05479=1125.587,-98.386,-46.172,179.563,4.444,148.866
C05480=1125.581,-98.137,-46.181,179.563,4.449,148.868
C05481=1125.576,-97.887,-46.190,179.563,4.454,148.869
C05482=1125.571,-97.637,-46.199,179.562,4.459,148.870
C05483=1125.565,-97.387,-46.208,179.562,4.463,148.871
C05484=1125.560,-97.138,-46.217,179.562,4.468,148.872
C05485=1125.554,-96.888,-46.226,179.562,4.474,148.873
C05486=1125.549,-96.638,-46.235,179.562,4.479,148.875
C05487=1125.543,-96.388,-46.244,179.561,4.484,148.876
